LIN {X 0,Y 420.94,Z 649.275,A -85,B 0,C 180,E1 -10152.356,E2 -10152.356} C_VEL
LIN {X 0,Y 419.985,Z 659.535,A -85,B 0,C 180,E1 -10153.721,E2 -10153.721} C_VEL
LIN {X 0,Y 419.053,Z 670.297,A -85,B 0,C 180,E1 -10155.428,E2 -10155.428} C_VEL
LIN {X 0,Y 418.282,Z 678.791,A -85,B 0,C 180,E1 -10157.037,E2 -10157.037} C_VEL
LIN {X 0,Y 417.855,Z 686.7,A -85,B 0,C 180,E1 -10158.846,E2 -10158.846} C_VEL
LIN {X 0,Y 417.37,Z 693.601,A -85,B 0,C 180,E1 -10160.794,E2 -10160.794} C_VEL
LIN {X 0,Y 417.15,Z 699.002,A -85,B 0,C 180,E1 -10162.739,E2 -10162.739} C_VEL
LIN {X 0,Y 417.07,Z 702.122,A -85,B 0,C 180,E1 -10164.196,E2 -10164.196} C_VEL
LIN {X 0,Y 416.971,Z 705.164,A -85,B 0,C 180,E1 -10166.133,E2 -10166.133} C_VEL
LIN {X 0,Y 417.064,Z 706.972,A -85,B 0,C 180,E1 -10168.067,E2 -10168.067} C_VEL
LIN {X 0,Y 417.001,Z 707.573,A -85,B 0,C 180,E1 -10169.999,E2 -10169.999} C_VEL
LIN {X 0,Y 417.065,Z 706.947,A -85,B 0,C 180,E1 -10171.93,E2 -10171.93} C_VEL
LIN {X 0,Y 416.99,Z 705.073,A -85,B 0,C 180,E1 -10173.864,E2 -10173.864} C_VEL
LIN {X 0,Y 417.068,Z 701.964,A -85,B 0,C 180,E1 -10175.801,E2 -10175.801} C_VEL
LIN {X 0,Y 417.23,Z 697.54,A -85,B 0,C 180,E1 -10177.743,E2 -10177.743} C_VEL
LIN {X 0,Y 417.436,Z 691.68,A -85,B 0,C 180,E1 -10179.691,E2 -10179.691} C_VEL
LIN {X 0,Y 417.936,Z 684.237,A -85,B 0,C 180,E1 -10181.64,E2 -10181.64} C_VEL
LIN {X 0,Y 418.477,Z 676.012,A -85,B 0,C 180,E1 -10183.394,E2 -10183.394} C_VEL
LIN {X 0,Y 419.269,Z 666.599,A -85,B 0,C 180,E1 -10185.058,E2 -10185.058} C_VEL
LIN {X 0,Y 420.141,Z 656.761,A -85,B 0,C 180,E1 -10186.52,E2 -10186.52} C_VEL
LIN {X 0,Y 421.138,Z 645.151,A -85,B 0,C 180,E1 -10187.97,E2 -10187.97} C_VEL
LIN {X 0,Y 422.119,Z 633.46,A -85,B 0,C 180,E1 -10189.196,E2 -10189.196} C_VEL
LIN {X 0,Y 423.228,Z 621.023,A -85,B 0,C 180,E1 -10190.28,E2 -10190.28} C_VEL
LIN {X 0,Y 424.236,Z 607.577,A -85,B 0,C 180,E1 -10191.245,E2 -10191.245} C_VEL
LIN {X 0,Y 425.287,Z 593.073,A -85,B 0,C 180,E1 -10192.071,E2 -10192.071} C_VEL
LIN {X 0,Y 426.147,Z 577.388,A -85,B 0,C 180,E1 -10192.75,E2 -10192.75} C_VEL
LIN {X 0,Y 426.824,Z 562.272,A -85,B 0,C 180,E1 -10193.205,E2 -10193.205} C_VEL
LIN {X 0,Y 429.831,Z 427.525,A -85,B 0,C 180,E1 -10195.772,E2 -10195.772} C_VEL
LIN {X 0,Y 423.925,Z 395.924,A -85,B 0,C 180,E1 -10196.788,E2 -10196.788} C_VEL
LIN {X 0,Y 424.456,Z 389.484,A -85,B 0,C 180,E1 -10197.84,E2 -10197.84} C_VEL
LIN {X 0,Y 421.951,Z 377.843,A -85,B 0,C 180,E1 -10199.991,E2 -10199.991} C_VEL
LIN {X 0,Y 418.225,Z 363.016,A -85,B 0,C 180,E1 -10202.888,E2 -10202.888} C_VEL
LIN {X 0,Y 418.23,Z 363.015,A -85,B 0,C 180,E1 -10206.023,E2 -10206.023} C_VEL
LIN {X 0,Y 418.195,Z 363.017,A -85,B 0,C 180,E1 -10209.371,E2 -10209.371} C_VEL
LIN {X 0,Y 418.202,Z 363.019,A -85,B 0,C 180,E1 -10212.317,E2 -10212.317} C_VEL
LIN {X 0,Y 418.223,Z 363.01,A -85,B 0,C 180,E1 -10215.107,E2 -10215.107} C_VEL
LIN {X 0,Y 418.208,Z 363.015,A -85,B 0,C 180,E1 -10217.763,E2 -10217.763} C_VEL
LIN {X 0,Y 418.221,Z 363.011,A -85,B 0,C 180,E1 -10221.555,E2 -10221.555} C_VEL
LIN {X 0,Y 418.244,Z 363.007,A -85,B 0,C 180,E1 -10225.158,E2 -10225.158} C_VEL
LIN {X 0,Y 418.232,Z 363.01,A -85,B 0,C 180,E1 -10227.471,E2 -10227.471} C_VEL
LIN {X 0,Y 418.245,Z 363.008,A -85,B 0,C 180,E1 -10230.897,E2 -10230.897} C_VEL
LIN {X 0,Y 418.204,Z 363.02,A -85,B 0,C 180,E1 -10234.092,E2 -10234.092} C_VEL
LIN {X 0,Y 418.213,Z 363.011,A -85,B 0,C 180,E1 -10237.263,E2 -10237.263} C_VEL
LIN {X 0,Y 418.268,Z 363.008,A -85,B 0,C 180,E1 -10240.364,E2 -10240.364} C_VEL
LIN {X 0,Y 418.264,Z 363.006,A -85,B 0,C 180,E1 -10243.403,E2 -10243.403} C_VEL
LIN {X 0,Y 418.331,Z 362.996,A -85,B 0,C 180,E1 -10246.999,E2 -10246.999} C_VEL
LIN {X 0,Y 418.319,Z 363.002,A -85,B 0,C 180,E1 -10250.328,E2 -10250.328} C_VEL
LIN {X 0,Y 418.427,Z 362.985,A -85,B 0,C 180,E1 -10253.248,E2 -10253.248} C_VEL
LIN {X 0,Y 418.302,Z 363,A -85,B 0,C 180,E1 -10255.181,E2 -10255.181} C_VEL
LIN {X 0,Y 418.517,Z 362.98,A -85,B 0,C 180,E1 -10258.076,E2 -10258.076} C_VEL
LIN {X 0,Y 418.526,Z 362.98,A -85,B 0,C 180,E1 -10260,E2 -10260} C_VEL
LIN {X 0,Y 418.453,Z 362.981,A -85,B 0,C 180,E1 -10262.888,E2 -10262.888} C_VEL
LIN {X 0,Y 418.425,Z 362.985,A -85,B 0,C 180,E1 -10266.512,E2 -10266.512} C_VEL
LIN {X 0,Y 418.354,Z 362.994,A -85,B 0,C 180,E1 -10268.696,E2 -10268.696} C_VEL
LIN {X 0,Y 418.339,Z 362.996,A -85,B 0,C 180,E1 -10272.615,E2 -10272.615} C_VEL
LIN {X 0,Y 418.237,Z 363.011,A -85,B 0,C 180,E1 -10275.597,E2 -10275.597} C_VEL
LIN {X 0,Y 418.255,Z 363.007,A -85,B 0,C 180,E1 -10278.618,E2 -10278.618} C_VEL
LIN {X 0,Y 418.22,Z 363.015,A -85,B 0,C 180,E1 -10281.697,E2 -10281.697} C_VEL
LIN {X 0,Y 418.231,Z 363.009,A -85,B 0,C 180,E1 -10284.853,E2 -10284.853} C_VEL
LIN {X 0,Y 418.195,Z 363.019,A -85,B 0,C 180,E1 -10288.071,E2 -10288.071} C_VEL
LIN {X 0,Y 418.227,Z 363.01,A -85,B 0,C 180,E1 -10291.021,E2 -10291.021} C_VEL
LIN {X 0,Y 418.236,Z 363.013,A -85,B 0,C 180,E1 -10293.679,E2 -10293.679} C_VEL
LIN {X 0,Y 418.222,Z 363.011,A -85,B 0,C 180,E1 -10297.226,E2 -10297.226} C_VEL
LIN {X 0,Y 418.197,Z 363.013,A -85,B 0,C 180,E1 -10300.869,E2 -10300.869} C_VEL
LIN {X 0,Y 418.193,Z 363.02,A -85,B 0,C 180,E1 -10303.73,E2 -10303.73} C_VEL
LIN {X 0,Y 418.192,Z 363.015,A -85,B 0,C 180,E1 -10306.449,E2 -10306.449} C_VEL
LIN {X 0,Y 418.199,Z 363.014,A -85,B 0,C 180,E1 -10309.135,E2 -10309.135} C_VEL
LIN {X 0,Y 418.228,Z 363.009,A -85,B 0,C 180,E1 -10312.777,E2 -10312.777} C_VEL
LIN {X 0,Y 418.232,Z 363.01,A -85,B 0,C 180,E1 -10316.324,E2 -10316.324} C_VEL
LIN {X 0,Y 418.237,Z 363.015,A -85,B 0,C 180,E1 -10319.729,E2 -10319.729} C_VEL
LIN {X 0,Y 418.207,Z 363.013,A -85,B 0,C 180,E1 -10323.018,E2 -10323.018} C_VEL
LIN {X 0,Y 418.254,Z 363.008,A -85,B 0,C 180,E1 -10326.219,E2 -10326.219} C_VEL
LIN {X 0,Y 418.248,Z 363.01,A -85,B 0,C 180,E1 -10329.339,E2 -10329.339} C_VEL
LIN {X 0,Y 418.278,Z 363.004,A -85,B 0,C 180,E1 -10332.397,E2 -10332.397} C_VEL
LIN {X 0,Y 418.301,Z 363.004,A -85,B 0,C 180,E1 -10335.405,E2 -10335.405} C_VEL
LIN {X 0,Y 418.314,Z 362.999,A -85,B 0,C 180,E1 -10338.371,E2 -10338.371} C_VEL
LIN {X 0,Y 418.448,Z 362.983,A -85,B 0,C 180,E1 -10342.28,E2 -10342.28} C_VEL
LIN {X 0,Y 418.473,Z 362.98,A -85,B 0,C 180,E1 -10344.218,E2 -10344.218} C_VEL
LIN {X 0,Y 418.536,Z 362.974,A -85,B 0,C 180,E1 -10348.077,E2 -10348.077} C_VEL
LIN {X 0,Y 418.546,Z 362.973,A -85,B 0,C 180,E1 -10350.001,E2 -10350.001} C_VEL
LIN {X 0,Y 418.476,Z 362.979,A -85,B 0,C 180,E1 -10352.889,E2 -10352.889} C_VEL
LIN {X 0,Y 418.489,Z 362.983,A -85,B 0,C 180,E1 -10355.784,E2 -10355.784} C_VEL
LIN {X 0,Y 418.382,Z 362.99,A -85,B 0,C 180,E1 -10358.697,E2 -10358.697} C_VEL
LIN {X 0,Y 418.319,Z 363.006,A -85,B 0,C 180,E1 -10361.632,E2 -10361.632} C_VEL
LIN {X 0,Y 418.327,Z 363.001,A -85,B 0,C 180,E1 -10363.305,E2 -10363.305} C_VEL
LIN {X 0,Y 417.621,Z 363.094,A -85,B 0,C 180,E1 -10364.108,E2 -10364.108} C_VEL
LIN {X 0,Y 414.724,Z 363.452,A -85,B 0,C 180,E1 -10365.413,E2 -10365.413} C_VEL
LIN {X 0,Y 412.302,Z 363.748,A -85,B 0,C 180,E1 -10366.466,E2 -10366.466} C_VEL
LIN {X 0,Y 411.278,Z 363.879,A -85,B 0,C 180,E1 -10367.281,E2 -10367.281} C_VEL
LIN {X 0,Y 411.203,Z 363.885,A -85,B 0,C 180,E1 -10367.557,E2 -10367.557} C_VEL
LIN {X 0,Y 411.202,Z 363.886,A -85,B 0,C 180,E1 -10371.035,E2 -10371.035} C_VEL
LIN {X 0,Y 411.198,Z 363.886,A -85,B 0,C 180,E1 -10374.218,E2 -10374.218} C_VEL
LIN {X 0,Y 411.178,Z 363.894,A -85,B 0,C 180,E1 -10377.485,E2 -10377.485} C_VEL
LIN {X 0,Y 411.203,Z 363.89,A -85,B 0,C 180,E1 -10379.714,E2 -10379.714} C_VEL
LIN {X 0,Y 411.213,Z 363.886,A -85,B 0,C 180,E1 -10383.156,E2 -10383.156} C_VEL
LIN {X 0,Y 411.198,Z 363.891,A -85,B 0,C 180,E1 -10386.553,E2 -10386.553} C_VEL
LIN {X 0,Y 411.202,Z 363.892,A -85,B 0,C 180,E1 -10389.725,E2 -10389.725} C_VEL
LIN {X 0,Y 411.218,Z 363.936,A -85,B 0,C 180,E1 -10391.576,E2 -10391.576} C_VEL
LIN {X 0,Y 413.441,Z 373.517,A -85,B 0,C 180,E1 -10393.635,E2 -10393.635} C_VEL
LIN {X 0,Y 422.18,Z 395.363,A -85,B 0,C 180,E1 -10394.659,E2 -10394.659} C_VEL
LIN {X 0,Y 423.567,Z 402.05,A -85,B 0,C 180,E1 -10394.884,E2 -10394.884} C_VEL
LIN {X 0,Y 420.269,Z 539.555,A -85,B 0,C 180,E1 -10397.564,E2 -10397.564} C_VEL
LIN {X 0,Y 419.622,Z 555.1,A -85,B 0,C 180,E1 -10398.059,E2 -10398.059} C_VEL
LIN {X 0,Y 418.811,Z 569.926,A -85,B 0,C 180,E1 -10398.723,E2 -10398.723} C_VEL
LIN {X 0,Y 417.84,Z 584.262,A -85,B 0,C 180,E1 -10399.562,E2 -10399.562} C_VEL
LIN {X 0,Y 416.764,Z 598.407,A -85,B 0,C 180,E1 -10400.607,E2 -10400.607} C_VEL
LIN {X 0,Y 415.718,Z 611,A -85,B 0,C 180,E1 -10401.744,E2 -10401.744} C_VEL
LIN {X 0,Y 414.639,Z 623.17,A -85,B 0,C 180,E1 -10403.068,E2 -10403.068} C_VEL
LIN {X 0,Y 413.561,Z 633.744,A -85,B 0,C 180,E1 -10404.436,E2 -10404.436} C_VEL
LIN {X 0,Y 412.613,Z 644.145,A -85,B 0,C 180,E1 -10406.038,E2 -10406.038} C_VEL
LIN {X 0,Y 411.827,Z 653.503,A -85,B 0,C 180,E1 -10407.771,E2 -10407.771} C_VEL
LIN {X 0,Y 411.09,Z 662.131,A -85,B 0,C 180,E1 -10409.713,E2 -10409.713} C_VEL
LIN {X 0,Y 410.679,Z 668.101,A -85,B 0,C 180,E1 -10411.369,E2 -10411.369} C_VEL
LIN {X 0,Y 410.394,Z 672.802,A -85,B 0,C 180,E1 -10412.938,E2 -10412.938} C_VEL
LIN {X 0,Y 410.122,Z 676.864,A -85,B 0,C 180,E1 -10414.633,E2 -10414.633} C_VEL
LIN {X 0,Y 409.878,Z 680.598,A -85,B 0,C 180,E1 -10416.773,E2 -10416.773} C_VEL
LIN {X 0,Y 409.789,Z 682.843,A -85,B 0,C 180,E1 -10418.89,E2 -10418.89} C_VEL
LIN {X 0,Y 409.82,Z 683.692,A -85,B 0,C 180,E1 -10420.984,E2 -10420.984} C_VEL
LIN {X 0,Y 409.799,Z 683.207,A -85,B 0,C 180,E1 -10423.049,E2 -10423.049} C_VEL
LIN {X 0,Y 409.883,Z 681.43,A -85,B 0,C 180,E1 -10425.096,E2 -10425.096} C_VEL
LIN {X 0,Y 410.102,Z 678.363,A -85,B 0,C 180,E1 -10427.127,E2 -10427.127} C_VEL
LIN {X 0,Y 410.393,Z 673.982,A -85,B 0,C 180,E1 -10429.142,E2 -10429.142} C_VEL
LIN {X 0,Y 410.823,Z 668.208,A -85,B 0,C 180,E1 -10431.143,E2 -10431.143} C_VEL
LIN {X 0,Y 411.487,Z 660.887,A -85,B 0,C 180,E1 -10433.133,E2 -10433.133} C_VEL
LIN {X 0,Y 412.241,Z 653.05,A -85,B 0,C 180,E1 -10434.865,E2 -10434.865} C_VEL
LIN {X 0,Y 413.188,Z 643.649,A -85,B 0,C 180,E1 -10436.587,E2 -10436.587} C_VEL
LIN {X 0,Y 414.249,Z 634.122,A -85,B 0,C 180,E1 -10438.055,E2 -10438.055} C_VEL
LIN {X 0,Y 415.254,Z 623.92,A -85,B 0,C 180,E1 -10439.396,E2 -10439.396} C_VEL
LIN {X 0,Y 416.508,Z 611.806,A -85,B 0,C 180,E1 -10440.725,E2 -10440.725} C_VEL
LIN {X 0,Y 417.817,Z 598.517,A -85,B 0,C 180,E1 -10441.928,E2 -10441.928} C_VEL
LIN {X 0,Y 418.892,Z 585.618,A -85,B 0,C 180,E1 -10442.885,E2 -10442.885} C_VEL
LIN {X 0,Y 420.035,Z 570.58,A -85,B 0,C 180,E1 -10443.777,E2 -10443.777} C_VEL
LIN {X 0,Y 420.971,Z 554.73,A -85,B 0,C 180,E1 -10444.488,E2 -10444.488} C_VEL
LIN {X 0,Y 421.672,Z 539.807,A -85,B 0,C 180,E1 -10444.96,E2 -10444.96} C_VEL
LIN {X 0,Y 425.402,Z 420.585,A -85,B 0,C 180,E1 -10447.467,E2 -10447.467} C_VEL
LIN {X 0,Y 425.949,Z 402.101,A -85,B 0,C 180,E1 -10447.883,E2 -10447.883} C_VEL
LIN {X 0,Y 424.63,Z 396.844,A -85,B 0,C 180,E1 -10448.128,E2 -10448.128} C_VEL
LIN {X 0,Y 418.317,Z 383.328,A -85,B 0,C 180,E1 -10449.044,E2 -10449.044} C_VEL
LIN {X 0,Y 414.737,Z 376.273,A -85,B 0,C 180,E1 -10449.587,E2 -10449.587} C_VEL
LIN {X 0,Y 411.965,Z 366.008,A -85,B 0,C 180,E1 -10452.312,E2 -10452.312} C_VEL
LIN {X 0,Y 411.308,Z 363.875,A -85,B 0,C 180,E1 -10452.98,E2 -10452.98} C_VEL
LIN {X 0,Y 411.259,Z 363.885,A -85,B 0,C 180,E1 -10455.868,E2 -10455.868} C_VEL
LIN {X 0,Y 411.224,Z 363.887,A -85,B 0,C 180,E1 -10458.948,E2 -10458.948} C_VEL
LIN {X 0,Y 411.204,Z 363.89,A -85,B 0,C 180,E1 -10462.64,E2 -10462.64} C_VEL
LIN {X 0,Y 411.188,Z 363.889,A -85,B 0,C 180,E1 -10465.296,E2 -10465.296} C_VEL
LIN {X 0,Y 411.176,Z 363.894,A -85,B 0,C 180,E1 -10468.593,E2 -10468.593} C_VEL
LIN {X 0,Y 411.167,Z 363.895,A -85,B 0,C 180,E1 -10471.997,E2 -10471.997} C_VEL
LIN {X 0,Y 411.205,Z 363.889,A -85,B 0,C 180,E1 -10474.876,E2 -10474.876} C_VEL
LIN {X 0,Y 411.192,Z 363.893,A -85,B 0,C 180,E1 -10478.165,E2 -10478.165} C_VEL
LIN {X 0,Y 411.162,Z 363.894,A -85,B 0,C 180,E1 -10481.807,E2 -10481.807} C_VEL
LIN {X 0,Y 411.176,Z 363.891,A -85,B 0,C 180,E1 -10485.508,E2 -10485.508} C_VEL
LIN {X 0,Y 411.148,Z 363.893,A -85,B 0,C 180,E1 -10488.774,E2 -10488.774} C_VEL
LIN {X 0,Y 411.18,Z 363.895,A -85,B 0,C 180,E1 -10492.023,E2 -10492.023} C_VEL
LIN {X 0,Y 411.225,Z 363.987,A -85,B 0,C 180,E1 -10495.025,E2 -10495.025} C_VEL
LIN {X 0,Y 414.638,Z 375.681,A -85,B 0,C 180,E1 -10497.939,E2 -10497.939} C_VEL
LIN {X 0,Y 417.107,Z 385.758,A -85,B 0,C 180,E1 -10500.193,E2 -10500.193} C_VEL
LIN {X 0,Y 418.526,Z 393.484,A -85,B 0,C 180,E1 -10501.786,E2 -10501.786} C_VEL
LIN {X 0,Y 422.778,Z 413.029,A -85,B 0,C 180,E1 -10502.685,E2 -10502.685} C_VEL
LIN {X 0,Y 425.409,Z 429.771,A -85,B 0,C 180,E1 -10503.323,E2 -10503.323} C_VEL
LIN {X 0,Y 422.133,Z 535.297,A -85,B 0,C 180,E1 -10505.534,E2 -10505.534} C_VEL
LIN {X 0,Y 421.243,Z 563.028,A -85,B 0,C 180,E1 -10506.134,E2 -10506.134} C_VEL
LIN {X 0,Y 420.294,Z 578.892,A -85,B 0,C 180,E1 -10506.661,E2 -10506.661} C_VEL
LIN {X 0,Y 419.23,Z 594.331,A -85,B 0,C 180,E1 -10507.384,E2 -10507.384} C_VEL
LIN {X 0,Y 418.005,Z 609.182,A -85,B 0,C 180,E1 -10508.29,E2 -10508.29} C_VEL
LIN {X 0,Y 416.732,Z 623.432,A -85,B 0,C 180,E1 -10509.386,E2 -10509.386} C_VEL
LIN {X 0,Y 415.387,Z 636.453,A -85,B 0,C 180,E1 -10510.606,E2 -10510.606} C_VEL
LIN {X 0,Y 414.126,Z 648.749,A -85,B 0,C 180,E1 -10511.998,E2 -10511.998} C_VEL
LIN {X 0,Y 413.12,Z 659.43,A -85,B 0,C 180,E1 -10513.443,E2 -10513.443} C_VEL
LIN {X 0,Y 412.127,Z 670.174,A -85,B 0,C 180,E1 -10515.178,E2 -10515.178} C_VEL
LIN {X 0,Y 411.239,Z 679.22,A -85,B 0,C 180,E1 -10516.935,E2 -10516.935} C_VEL
LIN {X 0,Y 410.818,Z 686.549,A -85,B 0,C 180,E1 -10518.653,E2 -10518.653} C_VEL
LIN {X 0,Y 410.316,Z 693.44,A -85,B 0,C 180,E1 -10520.634,E2 -10520.634} C_VEL
LIN {X 0,Y 410.093,Z 698.83,A -85,B 0,C 180,E1 -10522.614,E2 -10522.614} C_VEL
LIN {X 0,Y 409.978,Z 701.949,A -85,B 0,C 180,E1 -10524.095,E2 -10524.095} C_VEL
LIN {X 0,Y 409.888,Z 704.98,A -85,B 0,C 180,E1 -10526.066,E2 -10526.066} C_VEL
LIN {X 0,Y 409.973,Z 706.775,A -85,B 0,C 180,E1 -10528.034,E2 -10528.034} C_VEL
LIN {X 0,Y 409.923,Z 707.359,A -85,B 0,C 180,E1 -10529.999,E2 -10529.999} C_VEL
LIN {X 0,Y 409.992,Z 706.724,A -85,B 0,C 180,E1 -10531.963,E2 -10531.963} C_VEL
LIN {X 0,Y 409.907,Z 704.826,A -85,B 0,C 180,E1 -10533.931,E2 -10533.931} C_VEL
LIN {X 0,Y 409.975,Z 701.686,A -85,B 0,C 180,E1 -10535.902,E2 -10535.902} C_VEL
LIN {X 0,Y 410.152,Z 697.225,A -85,B 0,C 180,E1 -10537.877,E2 -10537.877} C_VEL
LIN {X 0,Y 410.364,Z 691.321,A -85,B 0,C 180,E1 -10539.86,E2 -10539.86} C_VEL
LIN {X 0,Y 410.862,Z 684.865,A -85,B 0,C 180,E1 -10541.593,E2 -10541.593} C_VEL
LIN {X 0,Y 411.384,Z 676.918,A -85,B 0,C 180,E1 -10543.355,E2 -10543.355} C_VEL
LIN {X 0,Y 412.179,Z 667.579,A -85,B 0,C 180,E1 -10545.07,E2 -10545.07} C_VEL
LIN {X 0,Y 413.071,Z 657.952,A -85,B 0,C 180,E1 -10546.556,E2 -10546.556} C_VEL
LIN {X 0,Y 414.067,Z 647.023,A -85,B 0,C 180,E1 -10547.977,E2 -10547.977} C_VEL
LIN {X 0,Y 415.201,Z 633.916,A -85,B 0,C 180,E1 -10549.4,E2 -10549.4} C_VEL
LIN {X 0,Y 416.477,Z 620.032,A -85,B 0,C 180,E1 -10550.624,E2 -10550.624} C_VEL
LIN {X 0,Y 417.525,Z 606.43,A -85,B 0,C 180,E1 -10551.604,E2 -10551.604} C_VEL
LIN {X 0,Y 418.655,Z 591.799,A -85,B 0,C 180,E1 -10552.433,E2 -10552.433} C_VEL
LIN {X 0,Y 419.49,Z 576.703,A -85,B 0,C 180,E1 -10553.086,E2 -10553.086} C_VEL
LIN {X 0,Y 420.179,Z 561.93,A -85,B 0,C 180,E1 -10553.535,E2 -10553.535} C_VEL
LIN {X 0,Y 423.328,Z 428.879,A -85,B 0,C 180,E1 -10556.121,E2 -10556.121} C_VEL
LIN {X 0,Y 417.205,Z 395.591,A -85,B 0,C 180,E1 -10557.235,E2 -10557.235} C_VEL
LIN {X 0,Y 417.492,Z 390.334,A -85,B 0,C 180,E1 -10558.12,E2 -10558.12} C_VEL
LIN {X 0,Y 414.952,Z 379.016,A -85,B 0,C 180,E1 -10560.256,E2 -10560.256} C_VEL
LIN {X 0,Y 411.185,Z 363.891,A -85,B 0,C 180,E1 -10563.265,E2 -10563.265} C_VEL
LIN {X 0,Y 411.18,Z 363.891,A -85,B 0,C 180,E1 -10566.55,E2 -10566.55} C_VEL
LIN {X 0,Y 411.158,Z 363.895,A -85,B 0,C 180,E1 -10569.719,E2 -10569.719} C_VEL
LIN {X 0,Y 411.154,Z 363.891,A -85,B 0,C 180,E1 -10573.134,E2 -10573.134} C_VEL
LIN {X 0,Y 411.152,Z 363.895,A -85,B 0,C 180,E1 -10575.881,E2 -10575.881} C_VEL
LIN {X 0,Y 411.135,Z 363.894,A -85,B 0,C 180,E1 -10578.773,E2 -10578.773} C_VEL
LIN {X 0,Y 411.169,Z 363.895,A -85,B 0,C 180,E1 -10582.024,E2 -10582.024} C_VEL
LIN {X 0,Y 411.192,Z 363.888,A -85,B 0,C 180,E1 -10585.665,E2 -10585.665} C_VEL
LIN {X 0,Y 411.175,Z 363.888,A -85,B 0,C 180,E1 -10589.151,E2 -10589.151} C_VEL
LIN {X 0,Y 411.158,Z 363.891,A -85,B 0,C 180,E1 -10591.406,E2 -10591.406} C_VEL
LIN {X 0,Y 411.173,Z 363.888,A -85,B 0,C 180,E1 -10594.941,E2 -10594.941} C_VEL
LIN {X 0,Y 411.188,Z 363.891,A -85,B 0,C 180,E1 -10597.913,E2 -10597.913} C_VEL
LIN {X 0,Y 411.2,Z 363.885,A -85,B 0,C 180,E1 -10601.051,E2 -10601.051} C_VEL
LIN {X 0,Y 411.195,Z 363.892,A -85,B 0,C 180,E1 -10604.13,E2 -10604.13} C_VEL
LIN {X 0,Y 411.288,Z 363.874,A -85,B 0,C 180,E1 -10607.165,E2 -10607.165} C_VEL
LIN {X 0,Y 411.272,Z 363.882,A -85,B 0,C 180,E1 -10610.161,E2 -10610.161} C_VEL
LIN {X 0,Y 411.376,Z 363.863,A -85,B 0,C 180,E1 -10613.132,E2 -10613.132} C_VEL
LIN {X 0,Y 411.274,Z 363.876,A -85,B 0,C 180,E1 -10615.099,E2 -10615.099} C_VEL
LIN {X 0,Y 411.486,Z 363.857,A -85,B 0,C 180,E1 -10618.043,E2 -10618.043} C_VEL
LIN {X 0,Y 411.361,Z 363.865,A -85,B 0,C 180,E1 -10620.979,E2 -10620.979} C_VEL
LIN {X 0,Y 411.411,Z 363.859,A -85,B 0,C 180,E1 -10622.938,E2 -10622.938} C_VEL
LIN {X 0,Y 411.375,Z 363.864,A -85,B 0,C 180,E1 -10626.509,E2 -10626.509} C_VEL
LIN {X 0,Y 411.294,Z 363.873,A -85,B 0,C 180,E1 -10628.847,E2 -10628.847} C_VEL
LIN {X 0,Y 411.26,Z 363.883,A -85,B 0,C 180,E1 -10631.834,E2 -10631.834} C_VEL
LIN {X 0,Y 411.217,Z 363.883,A -85,B 0,C 180,E1 -10634.855,E2 -10634.855} C_VEL
LIN {X 0,Y 411.216,Z 363.89,A -85,B 0,C 180,E1 -10637.917,E2 -10637.917} C_VEL
LIN {X 0,Y 411.182,Z 363.887,A -85,B 0,C 180,E1 -10641.035,E2 -10641.035} C_VEL
LIN {X 0,Y 411.179,Z 363.891,A -85,B 0,C 180,E1 -10644.219,E2 -10644.219} C_VEL
LIN {X 0,Y 411.134,Z 363.896,A -85,B 0,C 180,E1 -10647.487,E2 -10647.487} C_VEL
LIN {X 0,Y 411.184,Z 363.892,A -85,B 0,C 180,E1 -10649.714,E2 -10649.714} C_VEL
LIN {X 0,Y 411.196,Z 363.886,A -85,B 0,C 180,E1 -10653.157,E2 -10653.157} C_VEL
LIN {X 0,Y 411.178,Z 363.888,A -85,B 0,C 180,E1 -10656.553,E2 -10656.553} C_VEL
LIN {X 0,Y 411.157,Z 363.896,A -85,B 0,C 180,E1 -10659.722,E2 -10659.722} C_VEL
LIN {X 0,Y 411.153,Z 363.891,A -85,B 0,C 180,E1 -10663.137,E2 -10663.137} C_VEL
LIN {X 0,Y 411.155,Z 363.897,A -85,B 0,C 180,E1 -10665.883,E2 -10665.883} C_VEL
LIN {X 0,Y 411.14,Z 363.892,A -85,B 0,C 180,E1 -10668.776,E2 -10668.776} C_VEL
LIN {X 0,Y 411.175,Z 363.893,A -85,B 0,C 180,E1 -10672.027,E2 -10672.027} C_VEL
LIN {X 0,Y 411.193,Z 363.892,A -85,B 0,C 180,E1 -10675.667,E2 -10675.667} C_VEL
LIN {X 0,Y 411.184,Z 363.888,A -85,B 0,C 180,E1 -10679.154,E2 -10679.154} C_VEL
LIN {X 0,Y 411.172,Z 363.892,A -85,B 0,C 180,E1 -10681.408,E2 -10681.408} C_VEL
LIN {X 0,Y 411.185,Z 363.887,A -85,B 0,C 180,E1 -10684.943,E2 -10684.943} C_VEL
LIN {X 0,Y 411.201,Z 363.89,A -85,B 0,C 180,E1 -10687.915,E2 -10687.915} C_VEL
LIN {X 0,Y 411.217,Z 363.884,A -85,B 0,C 180,E1 -10691.053,E2 -10691.053} C_VEL
LIN {X 0,Y 411.253,Z 363.881,A -85,B 0,C 180,E1 -10694.133,E2 -10694.133} C_VEL
LIN {X 0,Y 411.304,Z 363.874,A -85,B 0,C 180,E1 -10697.167,E2 -10697.167} C_VEL
LIN {X 0,Y 411.289,Z 363.876,A -85,B 0,C 180,E1 -10700.163,E2 -10700.163} C_VEL
LIN {X 0,Y 411.392,Z 363.862,A -85,B 0,C 180,E1 -10703.133,E2 -10703.133} C_VEL
LIN {X 0,Y 411.289,Z 363.875,A -85,B 0,C 180,E1 -10705.1,E2 -10705.1} C_VEL
LIN {X 0,Y 411.505,Z 363.85,A -85,B 0,C 180,E1 -10708.044,E2 -10708.044} C_VEL
LIN {X 0,Y 411.38,Z 363.863,A -85,B 0,C 180,E1 -10710.98,E2 -10710.98} C_VEL
LIN {X 0,Y 411.434,Z 363.856,A -85,B 0,C 180,E1 -10712.939,E2 -10712.939} C_VEL
LIN {X 0,Y 411.434,Z 363.86,A -85,B 0,C 180,E1 -10715.884,E2 -10715.884} C_VEL
LIN {X 0,Y 411.323,Z 363.87,A -85,B 0,C 180,E1 -10718.847,E2 -10718.847} C_VEL
LIN {X 0,Y 411.288,Z 363.879,A -85,B 0,C 180,E1 -10721.834,E2 -10721.834} C_VEL
LIN {X 0,Y 411.237,Z 363.881,A -85,B 0,C 180,E1 -10724.855,E2 -10724.855} C_VEL
LIN {X 0,Y 411.203,Z 363.885,A -85,B 0,C 180,E1 -10727.557,E2 -10727.557} C_VEL
LIN {X 0,Y 410.554,Z 363.97,A -85,B 0,C 180,E1 -10728.375,E2 -10728.375} C_VEL
LIN {X 0,Y 407.698,Z 364.329,A -85,B 0,C 180,E1 -10729.705,E2 -10729.705} C_VEL
LIN {X 0,Y 405.272,Z 364.63,A -85,B 0,C 180,E1 -10730.778,E2 -10730.778} C_VEL
LIN {X 0,Y 404.233,Z 364.76,A -85,B 0,C 180,E1 -10731.608,E2 -10731.608} C_VEL
LIN {X 0,Y 404.151,Z 364.764,A -85,B 0,C 180,E1 -10731.89,E2 -10731.89} C_VEL
LIN {X 0,Y 404.158,Z 364.766,A -85,B 0,C 180,E1 -10735.278,E2 -10735.278} C_VEL
LIN {X 0,Y 404.157,Z 364.765,A -85,B 0,C 180,E1 -10739.138,E2 -10739.138} C_VEL
LIN {X 0,Y 404.148,Z 364.763,A -85,B 0,C 180,E1 -10742.622,E2 -10742.622} C_VEL
LIN {X 0,Y 404.187,Z 364.762,A -85,B 0,C 180,E1 -10745.19,E2 -10745.19} C_VEL
LIN {X 0,Y 404.149,Z 364.768,A -85,B 0,C 180,E1 -10748.759,E2 -10748.759} C_VEL
LIN {X 0,Y 404.153,Z 364.891,A -85,B 0,C 180,E1 -10751.238,E2 -10751.238} C_VEL
LIN {X 0,Y 406.285,Z 373.81,A -85,B 0,C 180,E1 -10753.183,E2 -10753.183} C_VEL
LIN {X 0,Y 415.848,Z 397.324,A -85,B 0,C 180,E1 -10754.318,E2 -10754.318} C_VEL
LIN {X 0,Y 417.046,Z 402.798,A -85,B 0,C 180,E1 -10754.51,E2 -10754.51} C_VEL
LIN {X 0,Y 413.581,Z 539.851,A -85,B 0,C 180,E1 -10757.24,E2 -10757.24} C_VEL
LIN {X 0,Y 412.9,Z 555.592,A -85,B 0,C 180,E1 -10757.752,E2 -10757.752} C_VEL
LIN {X 0,Y 412.048,Z 570.674,A -85,B 0,C 180,E1 -10758.446,E2 -10758.446} C_VEL
LIN {X 0,Y 410.996,Z 585.358,A -85,B 0,C 180,E1 -10759.33,E2 -10759.33} C_VEL
LIN {X 0,Y 409.922,Z 599.076,A -85,B 0,C 180,E1 -10760.37,E2 -10760.37} C_VEL
LIN {X 0,Y 408.734,Z 612.327,A -85,B 0,C 180,E1 -10761.599,E2 -10761.599} C_VEL
LIN {X 0,Y 407.689,Z 623.881,A -85,B 0,C 180,E1 -10762.889,E2 -10762.889} C_VEL
LIN {X 0,Y 406.559,Z 634.828,A -85,B 0,C 180,E1 -10764.339,E2 -10764.339} C_VEL
LIN {X 0,Y 405.574,Z 645.412,A -85,B 0,C 180,E1 -10766.024,E2 -10766.024} C_VEL
LIN {X 0,Y 404.793,Z 654.199,A -85,B 0,C 180,E1 -10767.7,E2 -10767.7} C_VEL
LIN {X 0,Y 404.037,Z 662.848,A -85,B 0,C 180,E1 -10769.705,E2 -10769.705} C_VEL
LIN {X 0,Y 403.588,Z 668.748,A -85,B 0,C 180,E1 -10771.387,E2 -10771.387} C_VEL
LIN {X 0,Y 403.278,Z 673.537,A -85,B 0,C 180,E1 -10773.056,E2 -10773.056} C_VEL
LIN {X 0,Y 402.969,Z 678.068,A -85,B 0,C 180,E1 -10775.083,E2 -10775.083} C_VEL
LIN {X 0,Y 402.806,Z 680.197,A -85,B 0,C 180,E1 -10776.34,E2 -10776.34} C_VEL
LIN {X 0,Y 402.704,Z 682.717,A -85,B 0,C 180,E1 -10778.5,E2 -10778.5} C_VEL
LIN {X 0,Y 402.737,Z 683.828,A -85,B 0,C 180,E1 -10780.636,E2 -10780.636} C_VEL
LIN {X 0,Y 402.682,Z 683.599,A -85,B 0,C 180,E1 -10782.74,E2 -10782.74} C_VEL
LIN {X 0,Y 402.776,Z 682.072,A -85,B 0,C 180,E1 -10784.827,E2 -10784.827} C_VEL
LIN {X 0,Y 402.965,Z 679.256,A -85,B 0,C 180,E1 -10786.895,E2 -10786.895} C_VEL
LIN {X 0,Y 403.293,Z 675.117,A -85,B 0,C 180,E1 -10788.948,E2 -10788.948} C_VEL
LIN {X 0,Y 403.708,Z 669.602,A -85,B 0,C 180,E1 -10790.986,E2 -10790.986} C_VEL
LIN {X 0,Y 404.378,Z 662.555,A -85,B 0,C 180,E1 -10793.012,E2 -10793.012} C_VEL
LIN {X 0,Y 405.164,Z 655.04,A -85,B 0,C 180,E1 -10794.775,E2 -10794.775} C_VEL
LIN {X 0,Y 406.135,Z 646.009,A -85,B 0,C 180,E1 -10796.527,E2 -10796.527} C_VEL
LIN {X 0,Y 407.412,Z 635.125,A -85,B 0,C 180,E1 -10798.27,E2 -10798.27} C_VEL
LIN {X 0,Y 408.6,Z 623.68,A -85,B 0,C 180,E1 -10799.795,E2 -10799.795} C_VEL
LIN {X 0,Y 410.039,Z 610.579,A -85,B 0,C 180,E1 -10801.227,E2 -10801.227} C_VEL
LIN {X 0,Y 411.399,Z 597.056,A -85,B 0,C 180,E1 -10802.447,E2 -10802.447} C_VEL
LIN {X 0,Y 412.598,Z 583.867,A -85,B 0,C 180,E1 -10803.418,E2 -10803.418} C_VEL
LIN {X 0,Y 413.71,Z 569.46,A -85,B 0,C 180,E1 -10804.262,E2 -10804.262} C_VEL
LIN {X 0,Y 414.635,Z 553.944,A -85,B 0,C 180,E1 -10804.953,E2 -10804.953} C_VEL
LIN {X 0,Y 415.376,Z 538.501,A -85,B 0,C 180,E1 -10805.431,E2 -10805.431} C_VEL
LIN {X 0,Y 419.277,Z 423.67,A -85,B 0,C 180,E1 -10807.906,E2 -10807.906} C_VEL
LIN {X 0,Y 419.998,Z 403.904,A -85,B 0,C 180,E1 -10808.35,E2 -10808.35} C_VEL
LIN {X 0,Y 418.921,Z 399.845,A -85,B 0,C 180,E1 -10808.549,E2 -10808.549} C_VEL
LIN {X 0,Y 413.107,Z 387.213,A -85,B 0,C 180,E1 -10809.437,E2 -10809.437} C_VEL
LIN {X 0,Y 407.601,Z 376.64,A -85,B 0,C 180,E1 -10810.314,E2 -10810.314} C_VEL
LIN {X 0,Y 404.865,Z 366.854,A -85,B 0,C 180,E1 -10813.042,E2 -10813.042} C_VEL
LIN {X 0,Y 404.229,Z 364.761,A -85,B 0,C 180,E1 -10813.735,E2 -10813.735} C_VEL
LIN {X 0,Y 404.208,Z 364.763,A -85,B 0,C 180,E1 -10817.192,E2 -10817.192} C_VEL
LIN {X 0,Y 404.169,Z 364.767,A -85,B 0,C 180,E1 -10820.351,E2 -10820.351} C_VEL
LIN {X 0,Y 404.154,Z 364.768,A -85,B 0,C 180,E1 -10823.575,E2 -10823.575} C_VEL
LIN {X 0,Y 404.109,Z 364.773,A -85,B 0,C 180,E1 -10826.883,E2 -10826.883} C_VEL
LIN {X 0,Y 404.146,Z 364.77,A -85,B 0,C 180,E1 -10830.285,E2 -10830.285} C_VEL
LIN {X 0,Y 404.141,Z 364.77,A -85,B 0,C 180,E1 -10833.812,E2 -10833.812} C_VEL
LIN {X 0,Y 404.134,Z 364.769,A -85,B 0,C 180,E1 -10836.873,E2 -10836.873} C_VEL
LIN {X 0,Y 404.121,Z 364.772,A -85,B 0,C 180,E1 -10840.074,E2 -10840.074} C_VEL
LIN {X 0,Y 404.143,Z 364.766,A -85,B 0,C 180,E1 -10843.081,E2 -10843.081} C_VEL
LIN {X 0,Y 404.123,Z 364.77,A -85,B 0,C 180,E1 -10845.921,E2 -10845.921} C_VEL
LIN {X 0,Y 404.103,Z 364.771,A -85,B 0,C 180,E1 -10848.632,E2 -10848.632} C_VEL
LIN {X 0,Y 404.136,Z 364.77,A -85,B 0,C 180,E1 -10851.495,E2 -10851.495} C_VEL
LIN {X 0,Y 404.156,Z 364.913,A -85,B 0,C 180,E1 -10854.294,E2 -10854.294} C_VEL
LIN {X 0,Y 407.365,Z 375.495,A -85,B 0,C 180,E1 -10857.081,E2 -10857.081} C_VEL
LIN {X 0,Y 409.882,Z 385.204,A -85,B 0,C 180,E1 -10859.376,E2 -10859.376} C_VEL
LIN {X 0,Y 411.663,Z 393.587,A -85,B 0,C 180,E1 -10861.154,E2 -10861.154} C_VEL
LIN {X 0,Y 413.251,Z 398.07,A -85,B 0,C 180,E1 -10861.431,E2 -10861.431} C_VEL
LIN {X 0,Y 417.178,Z 416.841,A -85,B 0,C 180,E1 -10862.298,E2 -10862.298} C_VEL
LIN {X 0,Y 419.34,Z 430.765,A -85,B 0,C 180,E1 -10862.838,E2 -10862.838} C_VEL
LIN {X 0,Y 415.755,Z 537.237,A -85,B 0,C 180,E1 -10865.133,E2 -10865.133} C_VEL
LIN {X 0,Y 414.859,Z 563.224,A -85,B 0,C 180,E1 -10865.71,E2 -10865.71} C_VEL
LIN {X 0,Y 413.787,Z 579.723,A -85,B 0,C 180,E1 -10866.276,E2 -10866.276} C_VEL
LIN {X 0,Y 412.71,Z 594.645,A -85,B 0,C 180,E1 -10866.999,E2 -10866.999} C_VEL
LIN {X 0,Y 411.415,Z 609.421,A -85,B 0,C 180,E1 -10867.924,E2 -10867.924} C_VEL
LIN {X 0,Y 410.083,Z 623.532,A -85,B 0,C 180,E1 -10869.036,E2 -10869.036} C_VEL
LIN {X 0,Y 408.676,Z 636.486,A -85,B 0,C 180,E1 -10870.275,E2 -10870.275} C_VEL
LIN {X 0,Y 407.397,Z 648.422,A -85,B 0,C 180,E1 -10871.65,E2 -10871.65} C_VEL
LIN {X 0,Y 406.277,Z 659.372,A -85,B 0,C 180,E1 -10873.156,E2 -10873.156} C_VEL
LIN {X 0,Y 405.202,Z 670.083,A -85,B 0,C 180,E1 -10874.919,E2 -10874.919} C_VEL
LIN {X 0,Y 404.383,Z 678.068,A -85,B 0,C 180,E1 -10876.48,E2 -10876.48} C_VEL
LIN {X 0,Y 403.897,Z 684.451,A -85,B 0,C 180,E1 -10877.946,E2 -10877.946} C_VEL
LIN {X 0,Y 403.479,Z 690.054,A -85,B 0,C 180,E1 -10879.46,E2 -10879.46} C_VEL
LIN {X 0,Y 403.119,Z 696.159,A -85,B 0,C 180,E1 -10881.477,E2 -10881.477} C_VEL
LIN {X 0,Y 402.976,Z 699.793,A -85,B 0,C 180,E1 -10882.986,E2 -10882.986} C_VEL
LIN {X 0,Y 402.857,Z 703.453,A -85,B 0,C 180,E1 -10884.994,E2 -10884.994} C_VEL
LIN {X 0,Y 402.803,Z 705.843,A -85,B 0,C 180,E1 -10886.998,E2 -10886.998} C_VEL
LIN {X 0,Y 402.862,Z 707.013,A -85,B 0,C 180,E1 -10888.999,E2 -10888.999} C_VEL
LIN {X 0,Y 402.862,Z 706.974,A -85,B 0,C 180,E1 -10890.998,E2 -10890.998} C_VEL
LIN {X 0,Y 402.902,Z 706.493,A -85,B 0,C 180,E1 -10891.998,E2 -10891.998} C_VEL
LIN {X 0,Y 402.826,Z 704.571,A -85,B 0,C 180,E1 -10894,E2 -10894} C_VEL
LIN {X 0,Y 402.897,Z 701.173,A -85,B 0,C 180,E1 -10896.128,E2 -10896.128} C_VEL
LIN {X 0,Y 403.069,Z 696.894,A -85,B 0,C 180,E1 -10898.017,E2 -10898.017} C_VEL
LIN {X 0,Y 403.303,Z 690.942,A -85,B 0,C 180,E1 -10900.034,E2 -10900.034} C_VEL
LIN {X 0,Y 403.795,Z 684.432,A -85,B 0,C 180,E1 -10901.799,E2 -10901.799} C_VEL
LIN {X 0,Y 404.354,Z 676.792,A -85,B 0,C 180,E1 -10903.518,E2 -10903.518} C_VEL
LIN {X 0,Y 405.242,Z 667.018,A -85,B 0,C 180,E1 -10905.334,E2 -10905.334} C_VEL
LIN {X 0,Y 406.178,Z 657.313,A -85,B 0,C 180,E1 -10906.846,E2 -10906.846} C_VEL
LIN {X 0,Y 407.256,Z 645.769,A -85,B 0,C 180,E1 -10908.354,E2 -10908.354} C_VEL
LIN {X 0,Y 408.422,Z 633.041,A -85,B 0,C 180,E1 -10909.735,E2 -10909.735} C_VEL
LIN {X 0,Y 409.602,Z 620.584,A -85,B 0,C 180,E1 -10910.855,E2 -10910.855} C_VEL
LIN {X 0,Y 410.686,Z 607.125,A -85,B 0,C 180,E1 -10911.85,E2 -10911.85} C_VEL
LIN {X 0,Y 411.802,Z 592.956,A -85,B 0,C 180,E1 -10912.682,E2 -10912.682} C_VEL
LIN {X 0,Y 412.761,Z 577.279,A -85,B 0,C 180,E1 -10913.385,E2 -10913.385} C_VEL
LIN {X 0,Y 413.527,Z 561.656,A -85,B 0,C 180,E1 -10913.87,E2 -10913.87} C_VEL
LIN {X 0,Y 416.734,Z 429.364,A -85,B 0,C 180,E1 -10916.502,E2 -10916.502} C_VEL
LIN {X 0,Y 410.498,Z 395.619,A -85,B 0,C 180,E1 -10917.635,E2 -10917.635} C_VEL
LIN {X 0,Y 410.561,Z 391.442,A -85,B 0,C 180,E1 -10918.359,E2 -10918.359} C_VEL
LIN {X 0,Y 407.434,Z 377.954,A -85,B 0,C 180,E1 -10920.964,E2 -10920.964} C_VEL
LIN {X 0,Y 404.16,Z 364.766,A -85,B 0,C 180,E1 -10923.628,E2 -10923.628} C_VEL
LIN {X 0,Y 404.123,Z 364.771,A -85,B 0,C 180,E1 -10926.873,E2 -10926.873} C_VEL
LIN {X 0,Y 404.107,Z 364.775,A -85,B 0,C 180,E1 -10930.073,E2 -10930.073} C_VEL
LIN {X 0,Y 404.133,Z 364.765,A -85,B 0,C 180,E1 -10933.081,E2 -10933.081} C_VEL
LIN {X 0,Y 404.133,Z 364.769,A -85,B 0,C 180,E1 -10935.924,E2 -10935.924} C_VEL
LIN {X 0,Y 404.09,Z 364.773,A -85,B 0,C 180,E1 -10938.632,E2 -10938.632} C_VEL
LIN {X 0,Y 404.125,Z 364.767,A -85,B 0,C 180,E1 -10941.494,E2 -10941.494} C_VEL
LIN {X 0,Y 404.17,Z 364.761,A -85,B 0,C 180,E1 -10944.983,E2 -10944.983} C_VEL
LIN {X 0,Y 404.126,Z 364.77,A -85,B 0,C 180,E1 -10948.441,E2 -10948.441} C_VEL
LIN {X 0,Y 404.135,Z 364.765,A -85,B 0,C 180,E1 -10950.862,E2 -10950.862} C_VEL
LIN {X 0,Y 404.138,Z 364.766,A -85,B 0,C 180,E1 -10954.722,E2 -10954.722} C_VEL
LIN {X 0,Y 404.152,Z 364.764,A -85,B 0,C 180,E1 -10957.507,E2 -10957.507} C_VEL
LIN {X 0,Y 404.145,Z 364.765,A -85,B 0,C 180,E1 -10960.707,E2 -10960.707} C_VEL
LIN {X 0,Y 404.166,Z 364.766,A -85,B 0,C 180,E1 -10963.846,E2 -10963.846} C_VEL
LIN {X 0,Y 404.268,Z 364.748,A -85,B 0,C 180,E1 -10966.939,E2 -10966.939} C_VEL
LIN {X 0,Y 404.238,Z 364.759,A -85,B 0,C 180,E1 -10969.988,E2 -10969.988} C_VEL
LIN {X 0,Y 404.326,Z 364.741,A -85,B 0,C 180,E1 -10973.012,E2 -10973.012} C_VEL
LIN {X 0,Y 404.246,Z 364.751,A -85,B 0,C 180,E1 -10975.013,E2 -10975.013} C_VEL
LIN {X 0,Y 404.455,Z 364.733,A -85,B 0,C 180,E1 -10978.009,E2 -10978.009} C_VEL
LIN {X 0,Y 404.331,Z 364.741,A -85,B 0,C 180,E1 -10980.996,E2 -10980.996} C_VEL
LIN {X 0,Y 404.371,Z 364.736,A -85,B 0,C 180,E1 -10982.989,E2 -10982.989} C_VEL
LIN {X 0,Y 404.327,Z 364.743,A -85,B 0,C 180,E1 -10986.505,E2 -10986.505} C_VEL
LIN {X 0,Y 404.243,Z 364.752,A -85,B 0,C 180,E1 -10989.002,E2 -10989.002} C_VEL
LIN {X 0,Y 404.234,Z 364.759,A -85,B 0,C 180,E1 -10992.042,E2 -10992.042} C_VEL
LIN {X 0,Y 404.161,Z 364.762,A -85,B 0,C 180,E1 -10995.12,E2 -10995.12} C_VEL
LIN {X 0,Y 404.18,Z 364.763,A -85,B 0,C 180,E1 -10998.24,E2 -10998.24} C_VEL
LIN {X 0,Y 404.124,Z 364.768,A -85,B 0,C 180,E1 -11001.421,E2 -11001.421} C_VEL
LIN {X 0,Y 404.123,Z 364.767,A -85,B 0,C 180,E1 -11004.67,E2 -11004.67} C_VEL
LIN {X 0,Y 404.091,Z 364.776,A -85,B 0,C 180,E1 -11008.008,E2 -11008.008} C_VEL
LIN {X 0,Y 404.132,Z 364.768,A -85,B 0,C 180,E1 -11010.287,E2 -11010.287} C_VEL
LIN {X 0,Y 404.133,Z 364.772,A -85,B 0,C 180,E1 -11013.814,E2 -11013.814} C_VEL
LIN {X 0,Y 404.12,Z 364.767,A -85,B 0,C 180,E1 -11016.875,E2 -11016.875} C_VEL
LIN {X 0,Y 404.107,Z 364.773,A -85,B 0,C 180,E1 -11020.076,E2 -11020.076} C_VEL
LIN {X 0,Y 404.133,Z 364.766,A -85,B 0,C 180,E1 -11023.083,E2 -11023.083} C_VEL
LIN {X 0,Y 404.112,Z 364.774,A -85,B 0,C 180,E1 -11025.924,E2 -11025.924} C_VEL
LIN {X 0,Y 404.094,Z 364.77,A -85,B 0,C 180,E1 -11028.634,E2 -11028.634} C_VEL
LIN {X 0,Y 404.131,Z 364.769,A -85,B 0,C 180,E1 -11031.497,E2 -11031.497} C_VEL
LIN {X 0,Y 404.17,Z 364.761,A -85,B 0,C 180,E1 -11034.985,E2 -11034.985} C_VEL
LIN {X 0,Y 404.134,Z 364.766,A -85,B 0,C 180,E1 -11038.444,E2 -11038.444} C_VEL
LIN {X 0,Y 404.147,Z 364.764,A -85,B 0,C 180,E1 -11040.864,E2 -11040.864} C_VEL
LIN {X 0,Y 404.15,Z 364.763,A -85,B 0,C 180,E1 -11044.724,E2 -11044.724} C_VEL
LIN {X 0,Y 404.164,Z 364.766,A -85,B 0,C 180,E1 -11047.51,E2 -11047.51} C_VEL
LIN {X 0,Y 404.161,Z 364.762,A -85,B 0,C 180,E1 -11050.709,E2 -11050.709} C_VEL
LIN {X 0,Y 404.22,Z 364.76,A -85,B 0,C 180,E1 -11053.85,E2 -11053.85} C_VEL
LIN {X 0,Y 404.284,Z 364.747,A -85,B 0,C 180,E1 -11056.941,E2 -11056.941} C_VEL
LIN {X 0,Y 404.255,Z 364.754,A -85,B 0,C 180,E1 -11059.99,E2 -11059.99} C_VEL
LIN {X 0,Y 404.342,Z 364.74,A -85,B 0,C 180,E1 -11063.013,E2 -11063.013} C_VEL
LIN {X 0,Y 404.26,Z 364.75,A -85,B 0,C 180,E1 -11065.015,E2 -11065.015} C_VEL
LIN {X 0,Y 404.474,Z 364.726,A -85,B 0,C 180,E1 -11068.01,E2 -11068.01} C_VEL
LIN {X 0,Y 404.351,Z 364.739,A -85,B 0,C 180,E1 -11070.997,E2 -11070.997} C_VEL
LIN {X 0,Y 404.394,Z 364.734,A -85,B 0,C 180,E1 -11072.99,E2 -11072.99} C_VEL
LIN {X 0,Y 404.382,Z 364.737,A -85,B 0,C 180,E1 -11075.987,E2 -11075.987} C_VEL
LIN {X 0,Y 404.27,Z 364.749,A -85,B 0,C 180,E1 -11079.003,E2 -11079.003} C_VEL
LIN {X 0,Y 404.261,Z 364.752,A -85,B 0,C 180,E1 -11082.043,E2 -11082.043} C_VEL
LIN {X 0,Y 404.182,Z 364.761,A -85,B 0,C 180,E1 -11085.12,E2 -11085.12} C_VEL
LIN {X 0,Y 404.172,Z 364.761,A -85,B 0,C 180,E1 -11088.241,E2 -11088.241} C_VEL
LIN {X 0,Y 404.165,Z 364.767,A -85,B 0,C 180,E1 -11091.419,E2 -11091.419} C_VEL
LIN {X 0,Y 404.151,Z 364.764,A -85,B 0,C 180,E1 -11091.89,E2 -11091.89} C_VEL
LIN {X 0,Y 403.495,Z 364.845,A -85,B 0,C 180,E1 -11092.721,E2 -11092.721} C_VEL
LIN {X 0,Y 400.659,Z 365.2,A -85,B 0,C 180,E1 -11094.072,E2 -11094.072} C_VEL
LIN {X 0,Y 398.24,Z 365.502,A -85,B 0,C 180,E1 -11095.163,E2 -11095.163} C_VEL
LIN {X 0,Y 397.181,Z 365.634,A -85,B 0,C 180,E1 -11096.007,E2 -11096.007} C_VEL
LIN {X 0,Y 397.085,Z 365.644,A -85,B 0,C 180,E1 -11096.293,E2 -11096.293} C_VEL
LIN {X 0,Y 397.105,Z 365.644,A -85,B 0,C 180,E1 -11099.864,E2 -11099.864} C_VEL
LIN {X 0,Y 397.125,Z 365.643,A -85,B 0,C 180,E1 -11103.719,E2 -11103.719} C_VEL
LIN {X 0,Y 397.097,Z 365.649,A -85,B 0,C 180,E1 -11107.209,E2 -11107.209} C_VEL
LIN {X 0,Y 397.127,Z 365.651,A -85,B 0,C 180,E1 -11110.849,E2 -11110.849} C_VEL
LIN {X 0,Y 399.043,Z 373.892,A -85,B 0,C 180,E1 -11112.694,E2 -11112.694} C_VEL
LIN {X 0,Y 409.645,Z 399.923,A -85,B 0,C 180,E1 -11113.988,E2 -11113.988} C_VEL
LIN {X 0,Y 410.505,Z 404.331,A -85,B 0,C 180,E1 -11114.139,E2 -11114.139} C_VEL
LIN {X 0,Y 406.927,Z 539.887,A -85,B 0,C 180,E1 -11116.899,E2 -11116.899} C_VEL
LIN {X 0,Y 406.263,Z 555.239,A -85,B 0,C 180,E1 -11117.403,E2 -11117.403} C_VEL
LIN {X 0,Y 405.352,Z 570.389,A -85,B 0,C 180,E1 -11118.103,E2 -11118.103} C_VEL
LIN {X 0,Y 404.305,Z 584.965,A -85,B 0,C 180,E1 -11118.988,E2 -11118.988} C_VEL
LIN {X 0,Y 403.194,Z 598.582,A -85,B 0,C 180,E1 -11120.025,E2 -11120.025} C_VEL
LIN {X 0,Y 402.055,Z 610.944,A -85,B 0,C 180,E1 -11121.168,E2 -11121.168} C_VEL
LIN {X 0,Y 400.833,Z 623.875,A -85,B 0,C 180,E1 -11122.62,E2 -11122.62} C_VEL
LIN {X 0,Y 399.717,Z 634.059,A -85,B 0,C 180,E1 -11123.98,E2 -11123.98} C_VEL
LIN {X 0,Y 398.68,Z 644.634,A -85,B 0,C 180,E1 -11125.66,E2 -11125.66} C_VEL
LIN {X 0,Y 397.828,Z 653.729,A -85,B 0,C 180,E1 -11127.397,E2 -11127.397} C_VEL
LIN {X 0,Y 397.034,Z 662.424,A -85,B 0,C 180,E1 -11129.409,E2 -11129.409} C_VEL
LIN {X 0,Y 396.51,Z 669.36,A -85,B 0,C 180,E1 -11131.408,E2 -11131.408} C_VEL
LIN {X 0,Y 396.177,Z 674.057,A -85,B 0,C 180,E1 -11133.105,E2 -11133.105} C_VEL
LIN {X 0,Y 395.897,Z 677.975,A -85,B 0,C 180,E1 -11134.873,E2 -11134.873} C_VEL
LIN {X 0,Y 395.686,Z 681.364,A -85,B 0,C 180,E1 -11136.998,E2 -11136.998} C_VEL
LIN {X 0,Y 395.582,Z 683.446,A -85,B 0,C 180,E1 -11139.186,E2 -11139.186} C_VEL
LIN {X 0,Y 395.593,Z 684.144,A -85,B 0,C 180,E1 -11141.35,E2 -11141.35} C_VEL
LIN {X 0,Y 395.617,Z 683.429,A -85,B 0,C 180,E1 -11143.598,E2 -11143.598} C_VEL
LIN {X 0,Y 395.736,Z 681.556,A -85,B 0,C 180,E1 -11145.603,E2 -11145.603} C_VEL
LIN {X 0,Y 396.036,Z 678.297,A -85,B 0,C 180,E1 -11147.704,E2 -11147.704} C_VEL
LIN {X 0,Y 396.357,Z 673.723,A -85,B 0,C 180,E1 -11149.786,E2 -11149.786} C_VEL
LIN {X 0,Y 396.937,Z 667.745,A -85,B 0,C 180,E1 -11151.857,E2 -11151.857} C_VEL
LIN {X 0,Y 397.726,Z 660.214,A -85,B 0,C 180,E1 -11153.914,E2 -11153.914} C_VEL
LIN {X 0,Y 398.619,Z 652.147,A -85,B 0,C 180,E1 -11155.702,E2 -11155.702} C_VEL
LIN {X 0,Y 399.734,Z 642.484,A -85,B 0,C 180,E1 -11157.481,E2 -11157.481} C_VEL
LIN {X 0,Y 400.868,Z 632.652,A -85,B 0,C 180,E1 -11158.995,E2 -11158.995} C_VEL
LIN {X 0,Y 402.305,Z 621.008,A -85,B 0,C 180,E1 -11160.5,E2 -11160.5} C_VEL
LIN {X 0,Y 403.762,Z 608.236,A -85,B 0,C 180,E1 -11161.87,E2 -11161.87} C_VEL
LIN {X 0,Y 405.042,Z 595.687,A -85,B 0,C 180,E1 -11162.984,E2 -11162.984} C_VEL
LIN {X 0,Y 406.336,Z 582.073,A -85,B 0,C 180,E1 -11163.967,E2 -11163.967} C_VEL
LIN {X 0,Y 407.395,Z 568.339,A -85,B 0,C 180,E1 -11164.762,E2 -11164.762} C_VEL
LIN {X 0,Y 408.426,Z 552.425,A -85,B 0,C 180,E1 -11165.461,E2 -11165.461} C_VEL
LIN {X 0,Y 409.169,Z 536.381,A -85,B 0,C 180,E1 -11165.946,E2 -11165.946} C_VEL
LIN {X 0,Y 412.739,Z 436.595,A -85,B 0,C 180,E1 -11168.144,E2 -11168.144} C_VEL
LIN {X 0,Y 414.011,Z 405.067,A -85,B 0,C 180,E1 -11168.868,E2 -11168.868} C_VEL
LIN {X 0,Y 412.537,Z 401.035,A -85,B 0,C 180,E1 -11169.117,E2 -11169.117} C_VEL
LIN {X 0,Y 406.647,Z 388.501,A -85,B 0,C 180,E1 -11170.054,E2 -11170.054} C_VEL
LIN {X 0,Y 400.5,Z 377.045,A -85,B 0,C 180,E1 -11171.083,E2 -11171.083} C_VEL
LIN {X 0,Y 397.925,Z 367.997,A -85,B 0,C 180,E1 -11173.735,E2 -11173.735} C_VEL
LIN {X 0,Y 397.162,Z 365.642,A -85,B 0,C 180,E1 -11174.54,E2 -11174.54} C_VEL
LIN {X 0,Y 397.149,Z 365.643,A -85,B 0,C 180,E1 -11177.507,E2 -11177.507} C_VEL
LIN {X 0,Y 397.108,Z 365.647,A -85,B 0,C 180,E1 -11180.729,E2 -11180.729} C_VEL
LIN {X 0,Y 397.112,Z 365.645,A -85,B 0,C 180,E1 -11184.019,E2 -11184.019} C_VEL
LIN {X 0,Y 397.07,Z 365.65,A -85,B 0,C 180,E1 -11187.399,E2 -11187.399} C_VEL
LIN {X 0,Y 397.101,Z 365.645,A -85,B 0,C 180,E1 -11189.862,E2 -11189.862} C_VEL
LIN {X 0,Y 397.116,Z 365.643,A -85,B 0,C 180,E1 -11193.273,E2 -11193.273} C_VEL
LIN {X 0,Y 397.096,Z 365.646,A -85,B 0,C 180,E1 -11196.995,E2 -11196.995} C_VEL
LIN {X 0,Y 397.058,Z 365.65,A -85,B 0,C 180,E1 -11200.437,E2 -11200.437} C_VEL
LIN {X 0,Y 397.089,Z 365.645,A -85,B 0,C 180,E1 -11203.65,E2 -11203.65} C_VEL
LIN {X 0,Y 397.093,Z 365.645,A -85,B 0,C 180,E1 -11206.522,E2 -11206.522} C_VEL
LIN {X 0,Y 397.087,Z 365.648,A -85,B 0,C 180,E1 -11210.418,E2 -11210.418} C_VEL
LIN {X 0,Y 397.132,Z 365.8,A -85,B 0,C 180,E1 -11213.482,E2 -11213.482} C_VEL
LIN {X 0,Y 400.418,Z 376.464,A -85,B 0,C 180,E1 -11216.456,E2 -11216.456} C_VEL
LIN {X 0,Y 403.148,Z 386.936,A -85,B 0,C 180,E1 -11219.033,E2 -11219.033} C_VEL
LIN {X 0,Y 404.494,Z 393.161,A -85,B 0,C 180,E1 -11220.407,E2 -11220.407} C_VEL
LIN {X 0,Y 407.562,Z 400.303,A -85,B 0,C 180,E1 -11220.93,E2 -11220.93} C_VEL
LIN {X 0,Y 411.326,Z 418.657,A -85,B 0,C 180,E1 -11221.803,E2 -11221.803} C_VEL
LIN {X 0,Y 413.297,Z 431.553,A -85,B 0,C 180,E1 -11222.331,E2 -11222.331} C_VEL
LIN {X 0,Y 409.528,Z 536.954,A -85,B 0,C 180,E1 -11224.661,E2 -11224.661} C_VEL
LIN {X 0,Y 408.51,Z 563.494,A -85,B 0,C 180,E1 -11225.273,E2 -11225.273} C_VEL
LIN {X 0,Y 407.336,Z 580.375,A -85,B 0,C 180,E1 -11225.873,E2 -11225.873} C_VEL
LIN {X 0,Y 406.154,Z 595.719,A -85,B 0,C 180,E1 -11226.641,E2 -11226.641} C_VEL
LIN {X 0,Y 404.849,Z 609.758,A -85,B 0,C 180,E1 -11227.547,E2 -11227.547} C_VEL
LIN {X 0,Y 403.443,Z 623.765,A -85,B 0,C 180,E1 -11228.675,E2 -11228.675} C_VEL
LIN {X 0,Y 401.97,Z 636.599,A -85,B 0,C 180,E1 -11229.931,E2 -11229.931} C_VEL
LIN {X 0,Y 400.688,Z 648.125,A -85,B 0,C 180,E1 -11231.289,E2 -11231.289} C_VEL
LIN {X 0,Y 399.435,Z 659.353,A -85,B 0,C 180,E1 -11232.858,E2 -11232.858} C_VEL
LIN {X 0,Y 398.289,Z 670.024,A -85,B 0,C 180,E1 -11234.651,E2 -11234.651} C_VEL
LIN {X 0,Y 397.33,Z 678.911,A -85,B 0,C 180,E1 -11236.444,E2 -11236.444} C_VEL
LIN {X 0,Y 396.755,Z 686.308,A -85,B 0,C 180,E1 -11238.245,E2 -11238.245} C_VEL
LIN {X 0,Y 396.193,Z 693.163,A -85,B 0,C 180,E1 -11240.297,E2 -11240.297} C_VEL
LIN {X 0,Y 395.939,Z 698.524,A -85,B 0,C 180,E1 -11242.348,E2 -11242.348} C_VEL
LIN {X 0,Y 395.82,Z 701.631,A -85,B 0,C 180,E1 -11243.883,E2 -11243.883} C_VEL
LIN {X 0,Y 395.731,Z 704.63,A -85,B 0,C 180,E1 -11245.925,E2 -11245.925} C_VEL
LIN {X 0,Y 395.766,Z 706.386,A -85,B 0,C 180,E1 -11247.963,E2 -11247.963} C_VEL
LIN {X 0,Y 395.775,Z 706.928,A -85,B 0,C 180,E1 -11249.998,E2 -11249.998} C_VEL
LIN {X 0,Y 395.799,Z 706.254,A -85,B 0,C 180,E1 -11252.034,E2 -11252.034} C_VEL
LIN {X 0,Y 395.747,Z 704.31,A -85,B 0,C 180,E1 -11254.072,E2 -11254.072} C_VEL
LIN {X 0,Y 395.818,Z 701.098,A -85,B 0,C 180,E1 -11256.114,E2 -11256.114} C_VEL
LIN {X 0,Y 395.982,Z 696.551,A -85,B 0,C 180,E1 -11258.161,E2 -11258.161} C_VEL
LIN {X 0,Y 396.245,Z 690.548,A -85,B 0,C 180,E1 -11260.215,E2 -11260.215} C_VEL
LIN {X 0,Y 396.746,Z 683.978,A -85,B 0,C 180,E1 -11262.012,E2 -11262.012} C_VEL
LIN {X 0,Y 397.388,Z 676.016,A -85,B 0,C 180,E1 -11263.811,E2 -11263.811} C_VEL
LIN {X 0,Y 398.287,Z 666.412,A -85,B 0,C 180,E1 -11265.609,E2 -11265.609} C_VEL
LIN {X 0,Y 399.28,Z 656.613,A -85,B 0,C 180,E1 -11267.145,E2 -11267.145} C_VEL
LIN {X 0,Y 400.412,Z 645.171,A -85,B 0,C 180,E1 -11268.654,E2 -11268.654} C_VEL
LIN {X 0,Y 401.522,Z 633.417,A -85,B 0,C 180,E1 -11269.955,E2 -11269.955} C_VEL
LIN {X 0,Y 402.878,Z 619.489,A -85,B 0,C 180,E1 -11271.22,E2 -11271.22} C_VEL
LIN {X 0,Y 404.04,Z 605.849,A -85,B 0,C 180,E1 -11272.228,E2 -11272.228} C_VEL
LIN {X 0,Y 405.193,Z 591.708,A -85,B 0,C 180,E1 -11273.058,E2 -11273.058} C_VEL
LIN {X 0,Y 406.082,Z 576.906,A -85,B 0,C 180,E1 -11273.725,E2 -11273.725} C_VEL
LIN {X 0,Y 406.888,Z 561.23,A -85,B 0,C 180,E1 -11274.217,E2 -11274.217} C_VEL
LIN {X 0,Y 410.206,Z 430.31,A -85,B 0,C 180,E1 -11276.878,E2 -11276.878} C_VEL
LIN {X 0,Y 403.777,Z 395.306,A -85,B 0,C 180,E1 -11278.1,E2 -11278.1} C_VEL
LIN {X 0,Y 403.327,Z 391.337,A -85,B 0,C 180,E1 -11278.836,E2 -11278.836} C_VEL
LIN {X 0,Y 399.741,Z 376.231,A -85,B 0,C 180,E1 -11281.831,E2 -11281.831} C_VEL
LIN {X 0,Y 397.116,Z 365.646,A -85,B 0,C 180,E1 -11284.059,E2 -11284.059} C_VEL
LIN {X 0,Y 397.079,Z 365.648,A -85,B 0,C 180,E1 -11287.206,E2 -11287.206} C_VEL
LIN {X 0,Y 397.045,Z 365.653,A -85,B 0,C 180,E1 -11290.436,E2 -11290.436} C_VEL
LIN {X 0,Y 397.087,Z 365.645,A -85,B 0,C 180,E1 -11293.648,E2 -11293.648} C_VEL
LIN {X 0,Y 397.085,Z 365.646,A -85,B 0,C 180,E1 -11296.521,E2 -11296.521} C_VEL
LIN {X 0,Y 397.073,Z 365.649,A -85,B 0,C 180,E1 -11300.418,E2 -11300.418} C_VEL
LIN {X 0,Y 397.081,Z 365.644,A -85,B 0,C 180,E1 -11303.003,E2 -11303.003} C_VEL
LIN {X 0,Y 397.105,Z 365.646,A -85,B 0,C 180,E1 -11306.281,E2 -11306.281} C_VEL
LIN {X 0,Y 397.085,Z 365.651,A -85,B 0,C 180,E1 -11310.136,E2 -11310.136} C_VEL
LIN {X 0,Y 397.06,Z 365.649,A -85,B 0,C 180,E1 -11313.737,E2 -11313.737} C_VEL
LIN {X 0,Y 397.084,Z 365.643,A -85,B 0,C 180,E1 -11317.084,E2 -11317.084} C_VEL
LIN {X 0,Y 397.13,Z 365.642,A -85,B 0,C 180,E1 -11320.352,E2 -11320.352} C_VEL
LIN {X 0,Y 397.112,Z 365.642,A -85,B 0,C 180,E1 -11323.551,E2 -11323.551} C_VEL
LIN {X 0,Y 397.214,Z 365.628,A -85,B 0,C 180,E1 -11326.702,E2 -11326.702} C_VEL
LIN {X 0,Y 397.199,Z 365.633,A -85,B 0,C 180,E1 -11329.809,E2 -11329.809} C_VEL
LIN {X 0,Y 397.278,Z 365.619,A -85,B 0,C 180,E1 -11332.887,E2 -11332.887} C_VEL
LIN {X 0,Y 397.217,Z 365.627,A -85,B 0,C 180,E1 -11334.925,E2 -11334.925} C_VEL
LIN {X 0,Y 397.424,Z 365.608,A -85,B 0,C 180,E1 -11337.973,E2 -11337.973} C_VEL
LIN {X 0,Y 397.302,Z 365.616,A -85,B 0,C 180,E1 -11341.014,E2 -11341.014} C_VEL
LIN {X 0,Y 397.305,Z 365.616,A -85,B 0,C 180,E1 -11343.042,E2 -11343.042} C_VEL
LIN {X 0,Y 397.284,Z 365.62,A -85,B 0,C 180,E1 -11346.498,E2 -11346.498} C_VEL
LIN {X 0,Y 397.214,Z 365.627,A -85,B 0,C 180,E1 -11349.163,E2 -11349.163} C_VEL
LIN {X 0,Y 397.2,Z 365.633,A -85,B 0,C 180,E1 -11352.259,E2 -11352.259} C_VEL
LIN {X 0,Y 397.11,Z 365.642,A -85,B 0,C 180,E1 -11355.395,E2 -11355.395} C_VEL
LIN {X 0,Y 397.137,Z 365.638,A -85,B 0,C 180,E1 -11358.575,E2 -11358.575} C_VEL
LIN {X 0,Y 397.081,Z 365.65,A -85,B 0,C 180,E1 -11361.82,E2 -11361.82} C_VEL
LIN {X 0,Y 397.09,Z 365.643,A -85,B 0,C 180,E1 -11365.137,E2 -11365.137} C_VEL
LIN {X 0,Y 397.051,Z 365.648,A -85,B 0,C 180,E1 -11368.55,E2 -11368.55} C_VEL
LIN {X 0,Y 397.071,Z 365.652,A -85,B 0,C 180,E1 -11371.838,E2 -11371.838} C_VEL
LIN {X 0,Y 397.113,Z 365.641,A -85,B 0,C 180,E1 -11374.495,E2 -11374.495} C_VEL
LIN {X 0,Y 397.079,Z 365.646,A -85,B 0,C 180,E1 -11378.278,E2 -11378.278} C_VEL
LIN {X 0,Y 397.042,Z 365.654,A -85,B 0,C 180,E1 -11381.978,E2 -11381.978} C_VEL
LIN {X 0,Y 397.076,Z 365.645,A -85,B 0,C 180,E1 -11385.071,E2 -11385.071} C_VEL
LIN {X 0,Y 397.044,Z 365.653,A -85,B 0,C 180,E1 -11388.025,E2 -11388.025} C_VEL
LIN {X 0,Y 397.083,Z 365.65,A -85,B 0,C 180,E1 -11391.725,E2 -11391.725} C_VEL
LIN {X 0,Y 397.114,Z 365.643,A -85,B 0,C 180,E1 -11395.508,E2 -11395.508} C_VEL
LIN {X 0,Y 397.073,Z 365.646,A -85,B 0,C 180,E1 -11399.119,E2 -11399.119} C_VEL
LIN {X 0,Y 397.059,Z 365.648,A -85,B 0,C 180,E1 -11402.253,E2 -11402.253} C_VEL
LIN {X 0,Y 397.1,Z 365.641,A -85,B 0,C 180,E1 -11404.867,E2 -11404.867} C_VEL
LIN {X 0,Y 397.093,Z 365.645,A -85,B 0,C 180,E1 -11408.183,E2 -11408.183} C_VEL
LIN {X 0,Y 397.156,Z 365.638,A -85,B 0,C 180,E1 -11411.428,E2 -11411.428} C_VEL
LIN {X 0,Y 397.178,Z 365.632,A -85,B 0,C 180,E1 -11414.61,E2 -11414.61} C_VEL
LIN {X 0,Y 397.219,Z 365.633,A -85,B 0,C 180,E1 -11417.744,E2 -11417.744} C_VEL
LIN {X 0,Y 397.235,Z 365.625,A -85,B 0,C 180,E1 -11420.839,E2 -11420.839} C_VEL
LIN {X 0,Y 397.323,Z 365.618,A -85,B 0,C 180,E1 -11423.909,E2 -11423.909} C_VEL
LIN {X 0,Y 397.442,Z 365.602,A -85,B 0,C 180,E1 -11427.975,E2 -11427.975} C_VEL
LIN {X 0,Y 397.322,Z 365.615,A -85,B 0,C 180,E1 -11431.015,E2 -11431.015} C_VEL
LIN {X 0,Y 397.328,Z 365.614,A -85,B 0,C 180,E1 -11433.043,E2 -11433.043} C_VEL
LIN {X 0,Y 397.333,Z 365.614,A -85,B 0,C 180,E1 -11436.094,E2 -11436.094} C_VEL
LIN {X 0,Y 397.24,Z 365.626,A -85,B 0,C 180,E1 -11439.164,E2 -11439.164} C_VEL
LIN {X 0,Y 397.224,Z 365.627,A -85,B 0,C 180,E1 -11442.259,E2 -11442.259} C_VEL
LIN {X 0,Y 397.131,Z 365.642,A -85,B 0,C 180,E1 -11445.395,E2 -11445.395} C_VEL
LIN {X 0,Y 397.12,Z 365.639,A -85,B 0,C 180,E1 -11448.577,E2 -11448.577} C_VEL
LIN {X 0,Y 397.109,Z 365.644,A -85,B 0,C 180,E1 -11451.88,E2 -11451.88} C_VEL
LIN {X 0,Y 397.102,Z 365.648,A -85,B 0,C 180,E1 -11455.496,E2 -11455.496} C_VEL
LIN {X 0,Y 397.085,Z 365.644,A -85,B 0,C 180,E1 -11456.293,E2 -11456.293} C_VEL
LIN {X 0,Y 396.392,Z 365.734,A -85,B 0,C 180,E1 -11457.139,E2 -11457.139} C_VEL
LIN {X 0,Y 393.539,Z 366.085,A -85,B 0,C 180,E1 -11458.516,E2 -11458.516} C_VEL
LIN {X 0,Y 391.138,Z 366.39,A -85,B 0,C 180,E1 -11459.629,E2 -11459.629} C_VEL
LIN {X 0,Y 390.104,Z 366.514,A -85,B 0,C 180,E1 -11460.488,E2 -11460.488} C_VEL
LIN {X 0,Y 390.017,Z 366.524,A -85,B 0,C 180,E1 -11460.78,E2 -11460.78} C_VEL
LIN {X 0,Y 390.075,Z 366.518,A -85,B 0,C 180,E1 -11464.025,E2 -11464.025} C_VEL
LIN {X 0,Y 390.047,Z 366.527,A -85,B 0,C 180,E1 -11467.551,E2 -11467.551} C_VEL
LIN {X 0,Y 390.097,Z 366.671,A -85,B 0,C 180,E1 -11470.511,E2 -11470.511} C_VEL
LIN {X 0,Y 391.931,Z 374.358,A -85,B 0,C 180,E1 -11472.219,E2 -11472.219} C_VEL
LIN {X 0,Y 403.461,Z 402.483,A -85,B 0,C 180,E1 -11473.65,E2 -11473.65} C_VEL
LIN {X 0,Y 404.025,Z 406.025,A -85,B 0,C 180,E1 -11473.768,E2 -11473.768} C_VEL
LIN {X 0,Y 400.287,Z 540.12,A -85,B 0,C 180,E1 -11476.553,E2 -11476.553} C_VEL
LIN {X 0,Y 399.564,Z 555.692,A -85,B 0,C 180,E1 -11477.075,E2 -11477.075} C_VEL
LIN {X 0,Y 398.659,Z 570.442,A -85,B 0,C 180,E1 -11477.769,E2 -11477.769} C_VEL
LIN {X 0,Y 397.612,Z 584.806,A -85,B 0,C 180,E1 -11478.652,E2 -11478.652} C_VEL
LIN {X 0,Y 396.39,Z 599.024,A -85,B 0,C 180,E1 -11479.753,E2 -11479.753} C_VEL
LIN {X 0,Y 395.115,Z 612.215,A -85,B 0,C 180,E1 -11481.007,E2 -11481.007} C_VEL
LIN {X 0,Y 393.964,Z 623.855,A -85,B 0,C 180,E1 -11482.338,E2 -11482.338} C_VEL
LIN {X 0,Y 392.765,Z 634.668,A -85,B 0,C 180,E1 -11483.808,E2 -11483.808} C_VEL
LIN {X 0,Y 391.766,Z 644.273,A -85,B 0,C 180,E1 -11485.361,E2 -11485.361} C_VEL
LIN {X 0,Y 390.903,Z 653.106,A -85,B 0,C 180,E1 -11487.053,E2 -11487.053} C_VEL
LIN {X 0,Y 390.19,Z 660.807,A -85,B 0,C 180,E1 -11488.812,E2 -11488.812} C_VEL
LIN {X 0,Y 389.548,Z 668.117,A -85,B 0,C 180,E1 -11490.848,E2 -11490.848} C_VEL
LIN {X 0,Y 389.195,Z 673.427,A -85,B 0,C 180,E1 -11492.687,E2 -11492.687} C_VEL
LIN {X 0,Y 388.857,Z 677.865,A -85,B 0,C 180,E1 -11494.648,E2 -11494.648} C_VEL
LIN {X 0,Y 388.62,Z 680.999,A -85,B 0,C 180,E1 -11496.555,E2 -11496.555} C_VEL
LIN {X 0,Y 388.505,Z 683.357,A -85,B 0,C 180,E1 -11498.789,E2 -11498.789} C_VEL
LIN {X 0,Y 388.534,Z 684.131,A -85,B 0,C 180,E1 -11500.155,E2 -11500.155} C_VEL
LIN {X 0,Y 388.487,Z 684.268,A -85,B 0,C 180,E1 -11502.089,E2 -11502.089} C_VEL
LIN {X 0,Y 388.561,Z 683.211,A -85,B 0,C 180,E1 -11504.257,E2 -11504.257} C_VEL
LIN {X 0,Y 388.735,Z 680.867,A -85,B 0,C 180,E1 -11506.406,E2 -11506.406} C_VEL
LIN {X 0,Y 389.087,Z 677.216,A -85,B 0,C 180,E1 -11508.539,E2 -11508.539} C_VEL
LIN {X 0,Y 389.498,Z 672.229,A -85,B 0,C 180,E1 -11510.654,E2 -11510.654} C_VEL
LIN {X 0,Y 390.195,Z 665.771,A -85,B 0,C 180,E1 -11512.757,E2 -11512.757} C_VEL
LIN {X 0,Y 391.109,Z 657.684,A -85,B 0,C 180,E1 -11514.845,E2 -11514.845} C_VEL
LIN {X 0,Y 392.155,Z 649.088,A -85,B 0,C 180,E1 -11516.661,E2 -11516.661} C_VEL
LIN {X 0,Y 393.348,Z 639.841,A -85,B 0,C 180,E1 -11518.297,E2 -11518.297} C_VEL
LIN {X 0,Y 394.597,Z 629.967,A -85,B 0,C 180,E1 -11519.775,E2 -11519.775} C_VEL
LIN {X 0,Y 396.078,Z 618.007,A -85,B 0,C 180,E1 -11521.271,E2 -11521.271} C_VEL
LIN {X 0,Y 397.545,Z 605.861,A -85,B 0,C 180,E1 -11522.533,E2 -11522.533} C_VEL
LIN {X 0,Y 398.909,Z 592.833,A -85,B 0,C 180,E1 -11523.661,E2 -11523.661} C_VEL
LIN {X 0,Y 400.34,Z 577.558,A -85,B 0,C 180,E1 -11524.72,E2 -11524.72} C_VEL
LIN {X 0,Y 401.564,Z 562.455,A -85,B 0,C 180,E1 -11525.523,E2 -11525.523} C_VEL
LIN {X 0,Y 402.471,Z 547.733,A -85,B 0,C 180,E1 -11526.108,E2 -11526.108} C_VEL
LIN {X 0,Y 403.157,Z 530.189,A -85,B 0,C 180,E1 -11526.575,E2 -11526.575} C_VEL
LIN {X 0,Y 406.498,Z 444.552,A -85,B 0,C 180,E1 -11528.504,E2 -11528.504} C_VEL
LIN {X 0,Y 408.126,Z 406.872,A -85,B 0,C 180,E1 -11529.384,E2 -11529.384} C_VEL
LIN {X 0,Y 403.125,Z 395.638,A -85,B 0,C 180,E1 -11530.22,E2 -11530.22} C_VEL
LIN {X 0,Y 397.176,Z 384.365,A -85,B 0,C 180,E1 -11531.224,E2 -11531.224} C_VEL
LIN {X 0,Y 393.435,Z 377.468,A -85,B 0,C 180,E1 -11531.907,E2 -11531.907} C_VEL
LIN {X 0,Y 390.859,Z 368.87,A -85,B 0,C 180,E1 -11534.58,E2 -11534.58} C_VEL
LIN {X 0,Y 390.151,Z 366.515,A -85,B 0,C 180,E1 -11535.408,E2 -11535.408} C_VEL
LIN {X 0,Y 390.107,Z 366.518,A -85,B 0,C 180,E1 -11538.922,E2 -11538.922} C_VEL
LIN {X 0,Y 390.04,Z 366.527,A -85,B 0,C 180,E1 -11542.234,E2 -11542.234} C_VEL
LIN {X 0,Y 390.055,Z 366.523,A -85,B 0,C 180,E1 -11545.721,E2 -11545.721} C_VEL
LIN {X 0,Y 390.028,Z 366.527,A -85,B 0,C 180,E1 -11549.112,E2 -11549.112} C_VEL
LIN {X 0,Y 390.045,Z 366.523,A -85,B 0,C 180,E1 -11552.721,E2 -11552.721} C_VEL
LIN {X 0,Y 390.045,Z 366.524,A -85,B 0,C 180,E1 -11555.821,E2 -11555.821} C_VEL
LIN {X 0,Y 390.039,Z 366.523,A -85,B 0,C 180,E1 -11559.211,E2 -11559.211} C_VEL
LIN {X 0,Y 390.032,Z 366.525,A -85,B 0,C 180,E1 -11562.371,E2 -11562.371} C_VEL
LIN {X 0,Y 390.043,Z 366.522,A -85,B 0,C 180,E1 -11565.353,E2 -11565.353} C_VEL
LIN {X 0,Y 390.017,Z 366.529,A -85,B 0,C 180,E1 -11568.183,E2 -11568.183} C_VEL
LIN {X 0,Y 390.057,Z 366.524,A -85,B 0,C 180,E1 -11570.902,E2 -11570.902} C_VEL
LIN {X 0,Y 390.049,Z 366.622,A -85,B 0,C 180,E1 -11572.569,E2 -11572.569} C_VEL
LIN {X 0,Y 392.971,Z 375.911,A -85,B 0,C 180,E1 -11575.353,E2 -11575.353} C_VEL
LIN {X 0,Y 395.576,Z 385.111,A -85,B 0,C 180,E1 -11577.791,E2 -11577.791} C_VEL
LIN {X 0,Y 397.36,Z 392.743,A -85,B 0,C 180,E1 -11579.606,E2 -11579.606} C_VEL
LIN {X 0,Y 402.067,Z 403.196,A -85,B 0,C 180,E1 -11580.441,E2 -11580.441} C_VEL
LIN {X 0,Y 405.526,Z 420.641,A -85,B 0,C 180,E1 -11581.3,E2 -11581.3} C_VEL
LIN {X 0,Y 407.342,Z 433.31,A -85,B 0,C 180,E1 -11581.821,E2 -11581.821} C_VEL
LIN {X 0,Y 403.376,Z 535.394,A -85,B 0,C 180,E1 -11584.142,E2 -11584.142} C_VEL
LIN {X 0,Y 402.33,Z 562.211,A -85,B 0,C 180,E1 -11584.764,E2 -11584.764} C_VEL
LIN {X 0,Y 401.282,Z 577.923,A -85,B 0,C 180,E1 -11585.316,E2 -11585.316} C_VEL
LIN {X 0,Y 400.127,Z 591.639,A -85,B 0,C 180,E1 -11585.972,E2 -11585.972} C_VEL
LIN {X 0,Y 398.855,Z 605.345,A -85,B 0,C 180,E1 -11586.815,E2 -11586.815} C_VEL
LIN {X 0,Y 397.352,Z 619.705,A -85,B 0,C 180,E1 -11587.922,E2 -11587.922} C_VEL
LIN {X 0,Y 395.777,Z 633.199,A -85,B 0,C 180,E1 -11589.196,E2 -11589.196} C_VEL
LIN {X 0,Y 394.419,Z 644.547,A -85,B 0,C 180,E1 -11590.481,E2 -11590.481} C_VEL
LIN {X 0,Y 393.235,Z 654.197,A -85,B 0,C 180,E1 -11591.773,E2 -11591.773} C_VEL
LIN {X 0,Y 391.992,Z 664.177,A -85,B 0,C 180,E1 -11593.328,E2 -11593.328} C_VEL
LIN {X 0,Y 390.893,Z 673.993,A -85,B 0,C 180,E1 -11595.154,E2 -11595.154} C_VEL
LIN {X 0,Y 390.042,Z 682.44,A -85,B 0,C 180,E1 -11597.047,E2 -11597.047} C_VEL
LIN {X 0,Y 389.413,Z 689.832,A -85,B 0,C 180,E1 -11599.075,E2 -11599.075} C_VEL
LIN {X 0,Y 388.981,Z 695.897,A -85,B 0,C 180,E1 -11601.164,E2 -11601.164} C_VEL
LIN {X 0,Y 388.82,Z 699.512,A -85,B 0,C 180,E1 -11602.73,E2 -11602.73} C_VEL
LIN {X 0,Y 388.663,Z 703.134,A -85,B 0,C 180,E1 -11604.811,E2 -11604.811} C_VEL
LIN {X 0,Y 388.613,Z 705.481,A -85,B 0,C 180,E1 -11606.888,E2 -11606.888} C_VEL
LIN {X 0,Y 388.703,Z 706.605,A -85,B 0,C 180,E1 -11608.962,E2 -11608.962} C_VEL
LIN {X 0,Y 388.722,Z 706.513,A -85,B 0,C 180,E1 -11611.034,E2 -11611.034} C_VEL
LIN {X 0,Y 388.625,Z 705.186,A -85,B 0,C 180,E1 -11613.108,E2 -11613.108} C_VEL
LIN {X 0,Y 388.676,Z 702.579,A -85,B 0,C 180,E1 -11615.186,E2 -11615.186} C_VEL
LIN {X 0,Y 388.826,Z 698.67,A -85,B 0,C 180,E1 -11617.267,E2 -11617.267} C_VEL
LIN {X 0,Y 389.027,Z 693.361,A -85,B 0,C 180,E1 -11619.356,E2 -11619.356} C_VEL
LIN {X 0,Y 389.54,Z 686.524,A -85,B 0,C 180,E1 -11621.445,E2 -11621.445} C_VEL
LIN {X 0,Y 390.069,Z 678.742,A -85,B 0,C 180,E1 -11623.362,E2 -11623.362} C_VEL
LIN {X 0,Y 390.913,Z 670.161,A -85,B 0,C 180,E1 -11625.109,E2 -11625.109} C_VEL
LIN {X 0,Y 392.025,Z 659.37,A -85,B 0,C 180,E1 -11626.935,E2 -11626.935} C_VEL
LIN {X 0,Y 393.22,Z 647.776,A -85,B 0,C 180,E1 -11628.561,E2 -11628.561} C_VEL
LIN {X 0,Y 394.487,Z 634.924,A -85,B 0,C 180,E1 -11630.055,E2 -11630.055} C_VEL
LIN {X 0,Y 395.74,Z 622.851,A -85,B 0,C 180,E1 -11631.212,E2 -11631.212} C_VEL
LIN {X 0,Y 396.879,Z 609.966,A -85,B 0,C 180,E1 -11632.24,E2 -11632.24} C_VEL
LIN {X 0,Y 398.161,Z 595.409,A -85,B 0,C 180,E1 -11633.169,E2 -11633.169} C_VEL
LIN {X 0,Y 399.145,Z 580.132,A -85,B 0,C 180,E1 -11633.922,E2 -11633.922} C_VEL
LIN {X 0,Y 399.979,Z 565.003,A -85,B 0,C 180,E1 -11634.455,E2 -11634.455} C_VEL
LIN {X 0,Y 400.712,Z 542.464,A -85,B 0,C 180,E1 -11634.961,E2 -11634.961} C_VEL
LIN {X 0,Y 403.694,Z 431.306,A -85,B 0,C 180,E1 -11637.258,E2 -11637.258} C_VEL
LIN {X 0,Y 396.926,Z 395.43,A -85,B 0,C 180,E1 -11638.53,E2 -11638.53} C_VEL
LIN {X 0,Y 394.719,Z 385.401,A -85,B 0,C 180,E1 -11640.492,E2 -11640.492} C_VEL
LIN {X 0,Y 391.094,Z 370.654,A -85,B 0,C 180,E1 -11643.542,E2 -11643.542} C_VEL
LIN {X 0,Y 390.08,Z 366.52,A -85,B 0,C 180,E1 -11644.458,E2 -11644.458} C_VEL
LIN {X 0,Y 390.026,Z 366.528,A -85,B 0,C 180,E1 -11647.779,E2 -11647.779} C_VEL
LIN {X 0,Y 390.007,Z 366.526,A -85,B 0,C 180,E1 -11650.813,E2 -11650.813} C_VEL
LIN {X 0,Y 390.041,Z 366.524,A -85,B 0,C 180,E1 -11653.884,E2 -11653.884} C_VEL
LIN {X 0,Y 390.039,Z 366.522,A -85,B 0,C 180,E1 -11656.787,E2 -11656.787} C_VEL
LIN {X 0,Y 389.997,Z 366.527,A -85,B 0,C 180,E1 -11659.553,E2 -11659.553} C_VEL
LIN {X 0,Y 390.025,Z 366.527,A -85,B 0,C 180,E1 -11662.449,E2 -11662.449} C_VEL
LIN {X 0,Y 390.055,Z 366.525,A -85,B 0,C 180,E1 -11666.044,E2 -11666.044} C_VEL
LIN {X 0,Y 390.03,Z 366.526,A -85,B 0,C 180,E1 -11669.869,E2 -11669.869} C_VEL
LIN {X 0,Y 390.016,Z 366.524,A -85,B 0,C 180,E1 -11673.225,E2 -11673.225} C_VEL
LIN {X 0,Y 390.05,Z 366.52,A -85,B 0,C 180,E1 -11676.764,E2 -11676.764} C_VEL
LIN {X 0,Y 390.088,Z 366.521,A -85,B 0,C 180,E1 -11679.982,E2 -11679.982} C_VEL
LIN {X 0,Y 390.091,Z 366.515,A -85,B 0,C 180,E1 -11683.246,E2 -11683.246} C_VEL
LIN {X 0,Y 390.18,Z 366.505,A -85,B 0,C 180,E1 -11686.561,E2 -11686.561} C_VEL
LIN {X 0,Y 390.15,Z 366.51,A -85,B 0,C 180,E1 -11689.623,E2 -11689.623} C_VEL
LIN {X 0,Y 390.231,Z 366.498,A -85,B 0,C 180,E1 -11692.758,E2 -11692.758} C_VEL
LIN {X 0,Y 390.189,Z 366.503,A -85,B 0,C 180,E1 -11694.833,E2 -11694.833} C_VEL
LIN {X 0,Y 390.391,Z 366.483,A -85,B 0,C 180,E1 -11697.937,E2 -11697.937} C_VEL
LIN {X 0,Y 390.273,Z 366.492,A -85,B 0,C 180,E1 -11701.032,E2 -11701.032} C_VEL
LIN {X 0,Y 390.241,Z 366.496,A -85,B 0,C 180,E1 -11703.097,E2 -11703.097} C_VEL
LIN {X 0,Y 390.244,Z 366.497,A -85,B 0,C 180,E1 -11706.489,E2 -11706.489} C_VEL
LIN {X 0,Y 390.172,Z 366.505,A -85,B 0,C 180,E1 -11709.33,E2 -11709.33} C_VEL
LIN {X 0,Y 390.181,Z 366.505,A -85,B 0,C 180,E1 -11713.439,E2 -11713.439} C_VEL
LIN {X 0,Y 390.094,Z 366.515,A -85,B 0,C 180,E1 -11717.289,E2 -11717.289} C_VEL
LIN {X 0,Y 390.075,Z 366.518,A -85,B 0,C 180,E1 -11720.471,E2 -11720.471} C_VEL
LIN {X 0,Y 390.048,Z 366.521,A -85,B 0,C 180,E1 -11723.354,E2 -11723.354} C_VEL
LIN {X 0,Y 390.017,Z 366.524,A -85,B 0,C 180,E1 -11726.776,E2 -11726.776} C_VEL
LIN {X 0,Y 390.025,Z 366.525,A -85,B 0,C 180,E1 -11730.301,E2 -11730.301} C_VEL
LIN {X 0,Y 390.058,Z 366.524,A -85,B 0,C 180,E1 -11734.026,E2 -11734.026} C_VEL
LIN {X 0,Y 390.027,Z 366.526,A -85,B 0,C 180,E1 -11737.551,E2 -11737.551} C_VEL
LIN {X 0,Y 390.006,Z 366.525,A -85,B 0,C 180,E1 -11740.816,E2 -11740.816} C_VEL
LIN {X 0,Y 390.042,Z 366.527,A -85,B 0,C 180,E1 -11743.887,E2 -11743.887} C_VEL
LIN {X 0,Y 390.039,Z 366.521,A -85,B 0,C 180,E1 -11746.79,E2 -11746.79} C_VEL
LIN {X 0,Y 390.002,Z 366.53,A -85,B 0,C 180,E1 -11749.556,E2 -11749.556} C_VEL
LIN {X 0,Y 390.031,Z 366.523,A -85,B 0,C 180,E1 -11752.452,E2 -11752.452} C_VEL
LIN {X 0,Y 390.059,Z 366.522,A -85,B 0,C 180,E1 -11756.047,E2 -11756.047} C_VEL
LIN {X 0,Y 390.039,Z 366.527,A -85,B 0,C 180,E1 -11759.872,E2 -11759.872} C_VEL
LIN {X 0,Y 390.028,Z 366.524,A -85,B 0,C 180,E1 -11763.228,E2 -11763.228} C_VEL
LIN {X 0,Y 390.062,Z 366.518,A -85,B 0,C 180,E1 -11766.767,E2 -11766.767} C_VEL
LIN {X 0,Y 390.102,Z 366.517,A -85,B 0,C 180,E1 -11769.985,E2 -11769.985} C_VEL
LIN {X 0,Y 390.138,Z 366.511,A -85,B 0,C 180,E1 -11773.25,E2 -11773.25} C_VEL
LIN {X 0,Y 390.195,Z 366.502,A -85,B 0,C 180,E1 -11776.563,E2 -11776.563} C_VEL
LIN {X 0,Y 390.167,Z 366.511,A -85,B 0,C 180,E1 -11779.624,E2 -11779.624} C_VEL
LIN {X 0,Y 390.248,Z 366.495,A -85,B 0,C 180,E1 -11782.759,E2 -11782.759} C_VEL
LIN {X 0,Y 390.202,Z 366.501,A -85,B 0,C 180,E1 -11784.835,E2 -11784.835} C_VEL
LIN {X 0,Y 390.41,Z 366.479,A -85,B 0,C 180,E1 -11787.938,E2 -11787.938} C_VEL
LIN {X 0,Y 390.292,Z 366.49,A -85,B 0,C 180,E1 -11791.033,E2 -11791.033} C_VEL
LIN {X 0,Y 390.264,Z 366.494,A -85,B 0,C 180,E1 -11793.098,E2 -11793.098} C_VEL
LIN {X 0,Y 390.287,Z 366.491,A -85,B 0,C 180,E1 -11796.204,E2 -11796.204} C_VEL
LIN {X 0,Y 390.197,Z 366.505,A -85,B 0,C 180,E1 -11799.33,E2 -11799.33} C_VEL
LIN {X 0,Y 390.176,Z 366.504,A -85,B 0,C 180,E1 -11802.484,E2 -11802.484} C_VEL
LIN {X 0,Y 390.073,Z 366.523,A -85,B 0,C 180,E1 -11805.681,E2 -11805.681} C_VEL
LIN {X 0,Y 390.081,Z 366.517,A -85,B 0,C 180,E1 -11808.925,E2 -11808.925} C_VEL
LIN {X 0,Y 390.048,Z 366.521,A -85,B 0,C 180,E1 -11812.235,E2 -11812.235} C_VEL
LIN {X 0,Y 390.056,Z 366.524,A -85,B 0,C 180,E1 -11815.723,E2 -11815.723} C_VEL
LIN {X 0,Y 390.034,Z 366.524,A -85,B 0,C 180,E1 -11819.113,E2 -11819.113} C_VEL
LIN {X 0,Y 390.017,Z 366.524,A -85,B 0,C 180,E1 -11820.78,E2 -11820.78} C_VEL
LIN {X 0,Y 389.344,Z 366.613,A -85,B 0,C 180,E1 -11821.642,E2 -11821.642} C_VEL
LIN {X 0,Y 386.498,Z 366.964,A -85,B 0,C 180,E1 -11823.043,E2 -11823.043} C_VEL
LIN {X 0,Y 384.101,Z 367.262,A -85,B 0,C 180,E1 -11824.176,E2 -11824.176} C_VEL
LIN {X 0,Y 383.082,Z 367.39,A -85,B 0,C 180,E1 -11825.052,E2 -11825.052} C_VEL
LIN {X 0,Y 383.004,Z 367.398,A -85,B 0,C 180,E1 -11825.349,E2 -11825.349} C_VEL
LIN {X 0,Y 382.992,Z 367.404,A -85,B 0,C 180,E1 -11828.604,E2 -11828.604} C_VEL
LIN {X 0,Y 383.028,Z 367.544,A -85,B 0,C 180,E1 -11830.129,E2 -11830.129} C_VEL
LIN {X 0,Y 384.688,Z 374.387,A -85,B 0,C 180,E1 -11831.71,E2 -11831.71} C_VEL
LIN {X 0,Y 397.183,Z 404.809,A -85,B 0,C 180,E1 -11833.295,E2 -11833.295} C_VEL
LIN {X 0,Y 397.54,Z 406.565,A -85,B 0,C 180,E1 -11833.359,E2 -11833.359} C_VEL
LIN {X 0,Y 393.637,Z 540.349,A -85,B 0,C 180,E1 -11836.201,E2 -11836.201} C_VEL
LIN {X 0,Y 392.882,Z 555.985,A -85,B 0,C 180,E1 -11836.737,E2 -11836.737} C_VEL
LIN {X 0,Y 391.89,Z 571.329,A -85,B 0,C 180,E1 -11837.478,E2 -11837.478} C_VEL
LIN {X 0,Y 390.727,Z 586.229,A -85,B 0,C 180,E1 -11838.424,E2 -11838.424} C_VEL
LIN {X 0,Y 389.538,Z 599.69,A -85,B 0,C 180,E1 -11839.495,E2 -11839.495} C_VEL
LIN {X 0,Y 388.31,Z 612.109,A -85,B 0,C 180,E1 -11840.693,E2 -11840.693} C_VEL
LIN {X 0,Y 386.989,Z 624.954,A -85,B 0,C 180,E1 -11842.198,E2 -11842.198} C_VEL
LIN {X 0,Y 385.754,Z 635.657,A -85,B 0,C 180,E1 -11843.692,E2 -11843.692} C_VEL
LIN {X 0,Y 384.637,Z 646.401,A -85,B 0,C 180,E1 -11845.498,E2 -11845.498} C_VEL
LIN {X 0,Y 383.65,Z 655.865,A -85,B 0,C 180,E1 -11847.424,E2 -11847.424} C_VEL
LIN {X 0,Y 382.891,Z 663.855,A -85,B 0,C 180,E1 -11849.406,E2 -11849.406} C_VEL
LIN {X 0,Y 382.343,Z 670.525,A -85,B 0,C 180,E1 -11851.45,E2 -11851.45} C_VEL
LIN {X 0,Y 381.996,Z 675.112,A -85,B 0,C 180,E1 -11853.208,E2 -11853.208} C_VEL
LIN {X 0,Y 381.696,Z 678.692,A -85,B 0,C 180,E1 -11854.945,E2 -11854.945} C_VEL
LIN {X 0,Y 381.486,Z 682.083,A -85,B 0,C 180,E1 -11857.239,E2 -11857.239} C_VEL
LIN {X 0,Y 381.413,Z 684.001,A -85,B 0,C 180,E1 -11859.506,E2 -11859.506} C_VEL
LIN {X 0,Y 381.407,Z 684.535,A -85,B 0,C 180,E1 -11861.744,E2 -11861.744} C_VEL
LIN {X 0,Y 381.463,Z 683.742,A -85,B 0,C 180,E1 -11863.957,E2 -11863.957} C_VEL
LIN {X 0,Y 381.607,Z 681.66,A -85,B 0,C 180,E1 -11866.147,E2 -11866.147} C_VEL
LIN {X 0,Y 381.994,Z 678.261,A -85,B 0,C 180,E1 -11868.323,E2 -11868.323} C_VEL
LIN {X 0,Y 382.413,Z 673.529,A -85,B 0,C 180,E1 -11870.479,E2 -11870.479} C_VEL
LIN {X 0,Y 383.102,Z 667.352,A -85,B 0,C 180,E1 -11872.622,E2 -11872.622} C_VEL
LIN {X 0,Y 384.059,Z 659.606,A -85,B 0,C 180,E1 -11874.75,E2 -11874.75} C_VEL
LIN {X 0,Y 385.101,Z 651.364,A -85,B 0,C 180,E1 -11876.599,E2 -11876.599} C_VEL
LIN {X 0,Y 386.474,Z 641.139,A -85,B 0,C 180,E1 -11878.489,E2 -11878.489} C_VEL
LIN {X 0,Y 387.78,Z 631.338,A -85,B 0,C 180,E1 -11880,E2 -11880} C_VEL
LIN {X 0,Y 389.368,Z 619.381,A -85,B 0,C 180,E1 -11881.551,E2 -11881.551} C_VEL
LIN {X 0,Y 391.073,Z 606.192,A -85,B 0,C 180,E1 -11882.961,E2 -11882.961} C_VEL
LIN {X 0,Y 392.503,Z 593.192,A -85,B 0,C 180,E1 -11884.107,E2 -11884.107} C_VEL
LIN {X 0,Y 394.018,Z 577.93,A -85,B 0,C 180,E1 -11885.181,E2 -11885.181} C_VEL
LIN {X 0,Y 395.309,Z 562.852,A -85,B 0,C 180,E1 -11885.995,E2 -11885.995} C_VEL
LIN {X 0,Y 396.251,Z 548.202,A -85,B 0,C 180,E1 -11886.594,E2 -11886.594} C_VEL
LIN {X 0,Y 396.992,Z 531.621,A -85,B 0,C 180,E1 -11887.054,E2 -11887.054} C_VEL
LIN {X 0,Y 400.572,Z 445.139,A -85,B 0,C 180,E1 -11889.051,E2 -11889.051} C_VEL
LIN {X 0,Y 402.229,Z 409.013,A -85,B 0,C 180,E1 -11889.926,E2 -11889.926} C_VEL
LIN {X 0,Y 397.462,Z 398.428,A -85,B 0,C 180,E1 -11890.754,E2 -11890.754} C_VEL
LIN {X 0,Y 392.158,Z 388.24,A -85,B 0,C 180,E1 -11891.703,E2 -11891.703} C_VEL
LIN {X 0,Y 386.355,Z 377.892,A -85,B 0,C 180,E1 -11892.808,E2 -11892.808} C_VEL
LIN {X 0,Y 383.94,Z 370.084,A -85,B 0,C 180,E1 -11895.392,E2 -11895.392} C_VEL
LIN {X 0,Y 383.084,Z 367.396,A -85,B 0,C 180,E1 -11896.383,E2 -11896.383} C_VEL
LIN {X 0,Y 383.064,Z 367.396,A -85,B 0,C 180,E1 -11899.283,E2 -11899.283} C_VEL
LIN {X 0,Y 382.993,Z 367.403,A -85,B 0,C 180,E1 -11902.665,E2 -11902.665} C_VEL
LIN {X 0,Y 382.987,Z 367.406,A -85,B 0,C 180,E1 -11906.13,E2 -11906.13} C_VEL
LIN {X 0,Y 382.979,Z 367.404,A -85,B 0,C 180,E1 -11909.701,E2 -11909.701} C_VEL
LIN {X 0,Y 383.003,Z 367.401,A -85,B 0,C 180,E1 -11913.4,E2 -11913.4} C_VEL
LIN {X 0,Y 383.025,Z 367.399,A -85,B 0,C 180,E1 -11916.161,E2 -11916.161} C_VEL
LIN {X 0,Y 382.988,Z 367.403,A -85,B 0,C 180,E1 -11919.58,E2 -11919.58} C_VEL
LIN {X 0,Y 383.01,Z 367.4,A -85,B 0,C 180,E1 -11922.778,E2 -11922.778} C_VEL
LIN {X 0,Y 382.992,Z 367.402,A -85,B 0,C 180,E1 -11925.787,E2 -11925.787} C_VEL
LIN {X 0,Y 382.964,Z 367.404,A -85,B 0,C 180,E1 -11928.8,E2 -11928.8} C_VEL
LIN {X 0,Y 382.994,Z 367.542,A -85,B 0,C 180,E1 -11931.595,E2 -11931.595} C_VEL
LIN {X 0,Y 386.101,Z 377.031,A -85,B 0,C 180,E1 -11934.64,E2 -11934.64} C_VEL
LIN {X 0,Y 388.639,Z 386.04,A -85,B 0,C 180,E1 -11937.144,E2 -11937.144} C_VEL
LIN {X 0,Y 390.203,Z 392.381,A -85,B 0,C 180,E1 -11938.736,E2 -11938.736} C_VEL
LIN {X 0,Y 396.709,Z 406.322,A -85,B 0,C 180,E1 -11939.949,E2 -11939.949} C_VEL
LIN {X 0,Y 400.181,Z 424.732,A -85,B 0,C 180,E1 -11940.868,E2 -11940.868} C_VEL
LIN {X 0,Y 401.454,Z 433.668,A -85,B 0,C 180,E1 -11941.259,E2 -11941.259} C_VEL
LIN {X 0,Y 397.172,Z 537.219,A -85,B 0,C 180,E1 -11943.672,E2 -11943.672} C_VEL
LIN {X 0,Y 396.044,Z 562.963,A -85,B 0,C 180,E1 -11944.299,E2 -11944.299} C_VEL
LIN {X 0,Y 394.861,Z 579.409,A -85,B 0,C 180,E1 -11944.904,E2 -11944.904} C_VEL
LIN {X 0,Y 393.586,Z 593.649,A -85,B 0,C 180,E1 -11945.625,E2 -11945.625} C_VEL
LIN {X 0,Y 392.147,Z 607.597,A -85,B 0,C 180,E1 -11946.529,E2 -11946.529} C_VEL
LIN {X 0,Y 390.591,Z 621.52,A -85,B 0,C 180,E1 -11947.658,E2 -11947.658} C_VEL
LIN {X 0,Y 388.988,Z 634.598,A -85,B 0,C 180,E1 -11948.954,E2 -11948.954} C_VEL
LIN {X 0,Y 387.436,Z 646.678,A -85,B 0,C 180,E1 -11950.391,E2 -11950.391} C_VEL
LIN {X 0,Y 386.229,Z 656.237,A -85,B 0,C 180,E1 -11951.723,E2 -11951.723} C_VEL
LIN {X 0,Y 384.806,Z 667.247,A -85,B 0,C 180,E1 -11953.554,E2 -11953.554} C_VEL
LIN {X 0,Y 383.678,Z 676.519,A -85,B 0,C 180,E1 -11955.411,E2 -11955.411} C_VEL
LIN {X 0,Y 382.861,Z 684.234,A -85,B 0,C 180,E1 -11957.273,E2 -11957.273} C_VEL
LIN {X 0,Y 382.391,Z 689.753,A -85,B 0,C 180,E1 -11958.872,E2 -11958.872} C_VEL
LIN {X 0,Y 381.904,Z 695.788,A -85,B 0,C 180,E1 -11960.999,E2 -11960.999} C_VEL
LIN {X 0,Y 381.729,Z 699.392,A -85,B 0,C 180,E1 -11962.594,E2 -11962.594} C_VEL
LIN {X 0,Y 381.575,Z 702.987,A -85,B 0,C 180,E1 -11964.715,E2 -11964.715} C_VEL
LIN {X 0,Y 381.523,Z 705.307,A -85,B 0,C 180,E1 -11966.831,E2 -11966.831} C_VEL
LIN {X 0,Y 381.617,Z 706.402,A -85,B 0,C 180,E1 -11968.943,E2 -11968.943} C_VEL
LIN {X 0,Y 381.636,Z 706.277,A -85,B 0,C 180,E1 -11971.054,E2 -11971.054} C_VEL
LIN {X 0,Y 381.536,Z 704.918,A -85,B 0,C 180,E1 -11973.166,E2 -11973.166} C_VEL
LIN {X 0,Y 381.584,Z 702.281,A -85,B 0,C 180,E1 -11975.282,E2 -11975.282} C_VEL
LIN {X 0,Y 381.732,Z 698.324,A -85,B 0,C 180,E1 -11977.403,E2 -11977.403} C_VEL
LIN {X 0,Y 381.968,Z 692.959,A -85,B 0,C 180,E1 -11979.53,E2 -11979.53} C_VEL
LIN {X 0,Y 382.509,Z 686.057,A -85,B 0,C 180,E1 -11981.658,E2 -11981.658} C_VEL
LIN {X 0,Y 383.03,Z 678.78,A -85,B 0,C 180,E1 -11983.477,E2 -11983.477} C_VEL
LIN {X 0,Y 383.948,Z 669.542,A -85,B 0,C 180,E1 -11985.39,E2 -11985.39} C_VEL
LIN {X 0,Y 384.939,Z 660.332,A -85,B 0,C 180,E1 -11986.983,E2 -11986.983} C_VEL
LIN {X 0,Y 386.169,Z 649.054,A -85,B 0,C 180,E1 -11988.624,E2 -11988.624} C_VEL
LIN {X 0,Y 387.459,Z 636.368,A -85,B 0,C 180,E1 -11990.158,E2 -11990.158} C_VEL
LIN {X 0,Y 388.878,Z 623.188,A -85,B 0,C 180,E1 -11991.465,E2 -11991.465} C_VEL
LIN {X 0,Y 390.057,Z 610.418,A -85,B 0,C 180,E1 -11992.51,E2 -11992.51} C_VEL
LIN {X 0,Y 391.403,Z 595.814,A -85,B 0,C 180,E1 -11993.466,E2 -11993.466} C_VEL
LIN {X 0,Y 392.437,Z 580.365,A -85,B 0,C 180,E1 -11994.249,E2 -11994.249} C_VEL
LIN {X 0,Y 393.299,Z 565.385,A -85,B 0,C 180,E1 -11994.793,E2 -11994.793} C_VEL
LIN {X 0,Y 394.048,Z 544.903,A -85,B 0,C 180,E1 -11995.271,E2 -11995.271} C_VEL
LIN {X 0,Y 397.188,Z 432.389,A -85,B 0,C 180,E1 -11997.647,E2 -11997.647} C_VEL
LIN {X 0,Y 390.796,Z 398.106,A -85,B 0,C 180,E1 -11998.885,E2 -11998.885} C_VEL
LIN {X 0,Y 389.681,Z 394.961,A -85,B 0,C 180,E1 -11999.064,E2 -11999.064} C_VEL
LIN {X 0,Y 386.171,Z 379.966,A -85,B 0,C 180,E1 -12002.134,E2 -12002.134} C_VEL
LIN {X 0,Y 383.046,Z 367.395,A -85,B 0,C 180,E1 -12004.863,E2 -12004.863} C_VEL
LIN {X 0,Y 382.971,Z 367.407,A -85,B 0,C 180,E1 -12008.602,E2 -12008.602} C_VEL
LIN {X 0,Y 382.95,Z 367.404,A -85,B 0,C 180,E1 -12011.349,E2 -12011.349} C_VEL
LIN {X 0,Y 382.983,Z 367.406,A -85,B 0,C 180,E1 -12014.302,E2 -12014.302} C_VEL
LIN {X 0,Y 382.999,Z 367.398,A -85,B 0,C 180,E1 -12017.239,E2 -12017.239} C_VEL
LIN {X 0,Y 382.972,Z 367.405,A -85,B 0,C 180,E1 -12020.418,E2 -12020.418} C_VEL
LIN {X 0,Y 383.004,Z 367.403,A -85,B 0,C 180,E1 -12024.042,E2 -12024.042} C_VEL
LIN {X 0,Y 382.974,Z 367.403,A -85,B 0,C 180,E1 -12027.577,E2 -12027.577} C_VEL
LIN {X 0,Y 382.962,Z 367.407,A -85,B 0,C 180,E1 -12030.298,E2 -12030.298} C_VEL
LIN {X 0,Y 382.988,Z 367.406,A -85,B 0,C 180,E1 -12034.044,E2 -12034.044} C_VEL
LIN {X 0,Y 382.974,Z 367.402,A -85,B 0,C 180,E1 -12037.333,E2 -12037.333} C_VEL
LIN {X 0,Y 383.041,Z 367.394,A -85,B 0,C 180,E1 -12040.716,E2 -12040.716} C_VEL
LIN {X 0,Y 383.005,Z 367.404,A -85,B 0,C 180,E1 -12044.024,E2 -12044.024} C_VEL
LIN {X 0,Y 383.121,Z 367.383,A -85,B 0,C 180,E1 -12047.284,E2 -12047.284} C_VEL
LIN {X 0,Y 383.127,Z 367.384,A -85,B 0,C 180,E1 -12050.498,E2 -12050.498} C_VEL
LIN {X 0,Y 383.224,Z 367.373,A -85,B 0,C 180,E1 -12053.683,E2 -12053.683} C_VEL
LIN {X 0,Y 383.357,Z 367.359,A -85,B 0,C 180,E1 -12057.899,E2 -12057.899} C_VEL
LIN {X 0,Y 383.244,Z 367.367,A -85,B 0,C 180,E1 -12061.051,E2 -12061.051} C_VEL
LIN {X 0,Y 383.357,Z 367.359,A -85,B 0,C 180,E1 -12062.102,E2 -12062.102} C_VEL
LIN {X 0,Y 383.209,Z 367.374,A -85,B 0,C 180,E1 -12066.476,E2 -12066.476} C_VEL
LIN {X 0,Y 383.123,Z 367.385,A -85,B 0,C 180,E1 -12069.503,E2 -12069.503} C_VEL
LIN {X 0,Y 383.112,Z 367.386,A -85,B 0,C 180,E1 -12073.537,E2 -12073.537} C_VEL
LIN {X 0,Y 383.044,Z 367.394,A -85,B 0,C 180,E1 -12077.438,E2 -12077.438} C_VEL
LIN {X 0,Y 383.016,Z 367.396,A -85,B 0,C 180,E1 -12080.648,E2 -12080.648} C_VEL
LIN {X 0,Y 382.997,Z 367.404,A -85,B 0,C 180,E1 -12083.81,E2 -12083.81} C_VEL
LIN {X 0,Y 382.957,Z 367.404,A -85,B 0,C 180,E1 -12087.31,E2 -12087.31} C_VEL
LIN {X 0,Y 382.97,Z 367.402,A -85,B 0,C 180,E1 -12090.92,E2 -12090.92} C_VEL
LIN {X 0,Y 383.003,Z 367.398,A -85,B 0,C 180,E1 -12094.67,E2 -12094.67} C_VEL
LIN {X 0,Y 382.982,Z 367.407,A -85,B 0,C 180,E1 -12097.904,E2 -12097.904} C_VEL
LIN {X 0,Y 382.951,Z 367.406,A -85,B 0,C 180,E1 -12101.352,E2 -12101.352} C_VEL
LIN {X 0,Y 382.984,Z 367.402,A -85,B 0,C 180,E1 -12104.304,E2 -12104.304} C_VEL
LIN {X 0,Y 382.988,Z 367.401,A -85,B 0,C 180,E1 -12107.24,E2 -12107.24} C_VEL
LIN {X 0,Y 382.978,Z 367.402,A -85,B 0,C 180,E1 -12110.421,E2 -12110.421} C_VEL
LIN {X 0,Y 383.008,Z 367.401,A -85,B 0,C 180,E1 -12114.045,E2 -12114.045} C_VEL
LIN {X 0,Y 382.981,Z 367.405,A -85,B 0,C 180,E1 -12117.58,E2 -12117.58} C_VEL
LIN {X 0,Y 382.972,Z 367.403,A -85,B 0,C 180,E1 -12120.301,E2 -12120.301} C_VEL
LIN {X 0,Y 382.999,Z 367.402,A -85,B 0,C 180,E1 -12124.047,E2 -12124.047} C_VEL
LIN {X 0,Y 382.986,Z 367.402,A -85,B 0,C 180,E1 -12127.336,E2 -12127.336} C_VEL
LIN {X 0,Y 383.057,Z 367.391,A -85,B 0,C 180,E1 -12130.718,E2 -12130.718} C_VEL
LIN {X 0,Y 383.08,Z 367.391,A -85,B 0,C 180,E1 -12134.028,E2 -12134.028} C_VEL
LIN {X 0,Y 383.137,Z 367.383,A -85,B 0,C 180,E1 -12137.286,E2 -12137.286} C_VEL
LIN {X 0,Y 383.143,Z 367.38,A -85,B 0,C 180,E1 -12140.499,E2 -12140.499} C_VEL
LIN {X 0,Y 383.236,Z 367.376,A -85,B 0,C 180,E1 -12143.685,E2 -12143.685} C_VEL
LIN {X 0,Y 383.376,Z 367.355,A -85,B 0,C 180,E1 -12147.9,E2 -12147.9} C_VEL
LIN {X 0,Y 383.263,Z 367.366,A -85,B 0,C 180,E1 -12151.052,E2 -12151.052} C_VEL
LIN {X 0,Y 383.377,Z 367.353,A -85,B 0,C 180,E1 -12152.103,E2 -12152.103} C_VEL
LIN {X 0,Y 383.244,Z 367.368,A -85,B 0,C 180,E1 -12156.318,E2 -12156.318} C_VEL
LIN {X 0,Y 383.148,Z 367.385,A -85,B 0,C 180,E1 -12159.504,E2 -12159.504} C_VEL
LIN {X 0,Y 383.131,Z 367.388,A -85,B 0,C 180,E1 -12163.537,E2 -12163.537} C_VEL
LIN {X 0,Y 383.06,Z 367.396,A -85,B 0,C 180,E1 -12167.436,E2 -12167.436} C_VEL
LIN {X 0,Y 383.037,Z 367.393,A -85,B 0,C 180,E1 -12170.649,E2 -12170.649} C_VEL
LIN {X 0,Y 383.015,Z 367.4,A -85,B 0,C 180,E1 -12173.81,E2 -12173.81} C_VEL
LIN {X 0,Y 382.987,Z 367.404,A -85,B 0,C 180,E1 -12177.309,E2 -12177.309} C_VEL
LIN {X 0,Y 382.989,Z 367.4,A -85,B 0,C 180,E1 -12180.919,E2 -12180.919} C_VEL
LIN {X 0,Y 383.025,Z 367.395,A -85,B 0,C 180,E1 -12184.669,E2 -12184.669} C_VEL
LIN {X 0,Y 383.004,Z 367.398,A -85,B 0,C 180,E1 -12185.349,E2 -12185.349} C_VEL
LIN {X 0,Y 382.336,Z 367.488,A -85,B 0,C 180,E1 -12185.934,E2 -12185.934} C_VEL
LIN {X 0,Y 379.501,Z 367.841,A -85,B 0,C 180,E1 -12186.85,E2 -12186.85} C_VEL
LIN {X 0,Y 376.633,Z 368.197,A -85,B 0,C 180,E1 -12187.778,E2 -12187.778} C_VEL
LIN {X 0,Y 375.939,Z 368.28,A -85,B 0,C 180,E1 -12188.379,E2 -12188.379} C_VEL
LIN {X 0,Y 375.98,Z 368.361,A -85,B 0,C 180,E1 -12189.72,E2 -12189.72} C_VEL
LIN {X 0,Y 377.511,Z 374.712,A -85,B 0,C 180,E1 -12191.192,E2 -12191.192} C_VEL
LIN {X 0,Y 390.151,Z 405.216,A -85,B 0,C 180,E1 -12192.841,E2 -12192.841} C_VEL
LIN {X 0,Y 391.051,Z 407.757,A -85,B 0,C 180,E1 -12192.961,E2 -12192.961} C_VEL
LIN {X 0,Y 386.983,Z 540.399,A -85,B 0,C 180,E1 -12195.841,E2 -12195.841} C_VEL
LIN {X 0,Y 386.186,Z 556.145,A -85,B 0,C 180,E1 -12196.389,E2 -12196.389} C_VEL
LIN {X 0,Y 385.199,Z 571.353,A -85,B 0,C 180,E1 -12197.136,E2 -12197.136} C_VEL
LIN {X 0,Y 384.015,Z 586.13,A -85,B 0,C 180,E1 -12198.087,E2 -12198.087} C_VEL
LIN {X 0,Y 382.794,Z 599.382,A -85,B 0,C 180,E1 -12199.151,E2 -12199.151} C_VEL
LIN {X 0,Y 381.365,Z 613.209,A -85,B 0,C 180,E1 -12200.516,E2 -12200.516} C_VEL
LIN {X 0,Y 380.131,Z 624.804,A -85,B 0,C 180,E1 -12201.899,E2 -12201.899} C_VEL
LIN {X 0,Y 378.737,Z 636.521,A -85,B 0,C 180,E1 -12203.572,E2 -12203.572} C_VEL
LIN {X 0,Y 377.603,Z 647.166,A -85,B 0,C 180,E1 -12205.412,E2 -12205.412} C_VEL
LIN {X 0,Y 376.634,Z 655.974,A -85,B 0,C 180,E1 -12207.238,E2 -12207.238} C_VEL
LIN {X 0,Y 375.844,Z 664.271,A -85,B 0,C 180,E1 -12209.337,E2 -12209.337} C_VEL
LIN {X 0,Y 375.292,Z 670.658,A -85,B 0,C 180,E1 -12211.328,E2 -12211.328} C_VEL
LIN {X 0,Y 374.904,Z 675.604,A -85,B 0,C 180,E1 -12213.262,E2 -12213.262} C_VEL
LIN {X 0,Y 374.607,Z 679.106,A -85,B 0,C 180,E1 -12215.031,E2 -12215.031} C_VEL
LIN {X 0,Y 374.429,Z 681.899,A -85,B 0,C 180,E1 -12216.888,E2 -12216.888} C_VEL
LIN {X 0,Y 374.301,Z 683.983,A -85,B 0,C 180,E1 -12219.099,E2 -12219.099} C_VEL
LIN {X 0,Y 374.339,Z 684.554,A -85,B 0,C 180,E1 -12220.248,E2 -12220.248} C_VEL
LIN {X 0,Y 374.309,Z 684.668,A -85,B 0,C 180,E1 -12222.517,E2 -12222.517} C_VEL
LIN {X 0,Y 374.394,Z 683.459,A -85,B 0,C 180,E1 -12224.763,E2 -12224.763} C_VEL
LIN {X 0,Y 374.699,Z 680.598,A -85,B 0,C 180,E1 -12227.251,E2 -12227.251} C_VEL
LIN {X 0,Y 375.035,Z 677.138,A -85,B 0,C 180,E1 -12229.199,E2 -12229.199} C_VEL
LIN {X 0,Y 375.572,Z 671.988,A -85,B 0,C 180,E1 -12231.39,E2 -12231.39} C_VEL
LIN {X 0,Y 376.435,Z 665.355,A -85,B 0,C 180,E1 -12233.568,E2 -12233.568} C_VEL
LIN {X 0,Y 377.396,Z 658.201,A -85,B 0,C 180,E1 -12235.46,E2 -12235.46} C_VEL
LIN {X 0,Y 378.575,Z 649.609,A -85,B 0,C 180,E1 -12237.34,E2 -12237.34} C_VEL
LIN {X 0,Y 380.135,Z 639.143,A -85,B 0,C 180,E1 -12239.233,E2 -12239.233} C_VEL
LIN {X 0,Y 381.526,Z 628.868,A -85,B 0,C 180,E1 -12240.791,E2 -12240.791} C_VEL
LIN {X 0,Y 383.282,Z 616.344,A -85,B 0,C 180,E1 -12242.364,E2 -12242.364} C_VEL
LIN {X 0,Y 385.09,Z 602.434,A -85,B 0,C 180,E1 -12243.793,E2 -12243.793} C_VEL
LIN {X 0,Y 386.671,Z 588.584,A -85,B 0,C 180,E1 -12244.952,E2 -12244.952} C_VEL
LIN {X 0,Y 388.14,Z 574.24,A -85,B 0,C 180,E1 -12245.911,E2 -12245.911} C_VEL
LIN {X 0,Y 389.399,Z 558.967,A -85,B 0,C 180,E1 -12246.7,E2 -12246.7} C_VEL
LIN {X 0,Y 390.456,Z 542.96,A -85,B 0,C 180,E1 -12247.292,E2 -12247.292} C_VEL
LIN {X 0,Y 395.805,Z 424.812,A -85,B 0,C 180,E1 -12250.14,E2 -12250.14} C_VEL
LIN {X 0,Y 396.436,Z 411.164,A -85,B 0,C 180,E1 -12250.485,E2 -12250.485} C_VEL
LIN {X 0,Y 391.543,Z 400.404,A -85,B 0,C 180,E1 -12251.387,E2 -12251.387} C_VEL
LIN {X 0,Y 384.322,Z 386.872,A -85,B 0,C 180,E1 -12252.753,E2 -12252.753} C_VEL
LIN {X 0,Y 380.656,Z 380.963,A -85,B 0,C 180,E1 -12253.47,E2 -12253.47} C_VEL
LIN {X 0,Y 379.224,Z 378.313,A -85,B 0,C 180,E1 -12253.804,E2 -12253.804} C_VEL
LIN {X 0,Y 377.035,Z 371.453,A -85,B 0,C 180,E1 -12256.236,E2 -12256.236} C_VEL
LIN {X 0,Y 376.033,Z 368.274,A -85,B 0,C 180,E1 -12257.496,E2 -12257.496} C_VEL
LIN {X 0,Y 375.984,Z 368.278,A -85,B 0,C 180,E1 -12260.831,E2 -12260.831} C_VEL
LIN {X 0,Y 375.964,Z 368.279,A -85,B 0,C 180,E1 -12264.283,E2 -12264.283} C_VEL
LIN {X 0,Y 375.922,Z 368.285,A -85,B 0,C 180,E1 -12267.864,E2 -12267.864} C_VEL
LIN {X 0,Y 375.958,Z 368.28,A -85,B 0,C 180,E1 -12270.692,E2 -12270.692} C_VEL
LIN {X 0,Y 375.961,Z 368.279,A -85,B 0,C 180,E1 -12274.111,E2 -12274.111} C_VEL
LIN {X 0,Y 375.951,Z 368.281,A -85,B 0,C 180,E1 -12276.741,E2 -12276.741} C_VEL
LIN {X 0,Y 375.941,Z 368.282,A -85,B 0,C 180,E1 -12279.96,E2 -12279.96} C_VEL
LIN {X 0,Y 375.927,Z 368.281,A -85,B 0,C 180,E1 -12283.766,E2 -12283.766} C_VEL
LIN {X 0,Y 375.936,Z 368.281,A -85,B 0,C 180,E1 -12286.81,E2 -12286.81} C_VEL
LIN {X 0,Y 375.964,Z 368.318,A -85,B 0,C 180,E1 -12290.474,E2 -12290.474} C_VEL
LIN {X 0,Y 378.32,Z 375.549,A -85,B 0,C 180,E1 -12293.016,E2 -12293.016} C_VEL
LIN {X 0,Y 380.692,Z 383.229,A -85,B 0,C 180,E1 -12295.391,E2 -12295.391} C_VEL
LIN {X 0,Y 383.055,Z 392.047,A -85,B 0,C 180,E1 -12297.795,E2 -12297.795} C_VEL
LIN {X 0,Y 389.677,Z 405.53,A -85,B 0,C 180,E1 -12299.096,E2 -12299.096} C_VEL
LIN {X 0,Y 391.598,Z 410.38,A -85,B 0,C 180,E1 -12299.48,E2 -12299.48} C_VEL
LIN {X 0,Y 394.882,Z 428.859,A -85,B 0,C 180,E1 -12300.424,E2 -12300.424} C_VEL
LIN {X 0,Y 395.637,Z 435.429,A -85,B 0,C 180,E1 -12300.7,E2 -12300.7} C_VEL
LIN {X 0,Y 391.354,Z 531.071,A -85,B 0,C 180,E1 -12302.998,E2 -12302.998} C_VEL
LIN {X 0,Y 389.947,Z 562.318,A -85,B 0,C 180,E1 -12303.759,E2 -12303.759} C_VEL
LIN {X 0,Y 388.739,Z 578.342,A -85,B 0,C 180,E1 -12304.356,E2 -12304.356} C_VEL
LIN {X 0,Y 387.422,Z 592.148,A -85,B 0,C 180,E1 -12305.053,E2 -12305.053} C_VEL
LIN {X 0,Y 385.873,Z 606.746,A -85,B 0,C 180,E1 -12306.007,E2 -12306.007} C_VEL
LIN {X 0,Y 384.458,Z 619.1,A -85,B 0,C 180,E1 -12306.998,E2 -12306.998} C_VEL
LIN {X 0,Y 382.694,Z 632.56,A -85,B 0,C 180,E1 -12308.308,E2 -12308.308} C_VEL
LIN {X 0,Y 380.995,Z 644.908,A -85,B 0,C 180,E1 -12309.764,E2 -12309.764} C_VEL
LIN {X 0,Y 379.419,Z 656.488,A -85,B 0,C 180,E1 -12311.408,E2 -12311.408} C_VEL
LIN {X 0,Y 377.928,Z 667.287,A -85,B 0,C 180,E1 -12313.246,E2 -12313.246} C_VEL
LIN {X 0,Y 376.744,Z 676.529,A -85,B 0,C 180,E1 -12315.136,E2 -12315.136} C_VEL
LIN {X 0,Y 375.884,Z 684.231,A -85,B 0,C 180,E1 -12317.033,E2 -12317.033} C_VEL
LIN {X 0,Y 375.167,Z 691.382,A -85,B 0,C 180,E1 -12319.202,E2 -12319.202} C_VEL
LIN {X 0,Y 374.786,Z 697.005,A -85,B 0,C 180,E1 -12321.371,E2 -12321.371} C_VEL
LIN {X 0,Y 374.563,Z 701.231,A -85,B 0,C 180,E1 -12323.534,E2 -12323.534} C_VEL
LIN {X 0,Y 374.483,Z 704.148,A -85,B 0,C 180,E1 -12325.693,E2 -12325.693} C_VEL
LIN {X 0,Y 374.459,Z 705.82,A -85,B 0,C 180,E1 -12327.847,E2 -12327.847} C_VEL
LIN {X 0,Y 374.551,Z 706.272,A -85,B 0,C 180,E1 -12329.998,E2 -12329.998} C_VEL
LIN {X 0,Y 374.492,Z 705.492,A -85,B 0,C 180,E1 -12332.149,E2 -12332.149} C_VEL
LIN {X 0,Y 374.518,Z 703.472,A -85,B 0,C 180,E1 -12334.303,E2 -12334.303} C_VEL
LIN {X 0,Y 374.568,Z 700.142,A -85,B 0,C 180,E1 -12336.462,E2 -12336.462} C_VEL
LIN {X 0,Y 374.757,Z 695.441,A -85,B 0,C 180,E1 -12338.627,E2 -12338.627} C_VEL
LIN {X 0,Y 375.119,Z 689.261,A -85,B 0,C 180,E1 -12340.797,E2 -12340.797} C_VEL
LIN {X 0,Y 375.816,Z 681.448,A -85,B 0,C 180,E1 -12342.966,E2 -12342.966} C_VEL
LIN {X 0,Y 376.604,Z 673.027,A -85,B 0,C 180,E1 -12344.866,E2 -12344.866} C_VEL
LIN {X 0,Y 377.653,Z 662.889,A -85,B 0,C 180,E1 -12346.763,E2 -12346.763} C_VEL
LIN {X 0,Y 378.997,Z 651.186,A -85,B 0,C 180,E1 -12348.568,E2 -12348.568} C_VEL
LIN {X 0,Y 380.268,Z 638.932,A -85,B 0,C 180,E1 -12350.132,E2 -12350.132} C_VEL
LIN {X 0,Y 381.757,Z 626.326,A -85,B 0,C 180,E1 -12351.46,E2 -12351.46} C_VEL
LIN {X 0,Y 383.095,Z 612.535,A -85,B 0,C 180,E1 -12352.657,E2 -12352.657} C_VEL
LIN {X 0,Y 384.47,Z 598.386,A -85,B 0,C 180,E1 -12353.639,E2 -12353.639} C_VEL
LIN {X 0,Y 385.599,Z 583.226,A -85,B 0,C 180,E1 -12354.461,E2 -12354.461} C_VEL
LIN {X 0,Y 386.578,Z 567.645,A -85,B 0,C 180,E1 -12355.074,E2 -12355.074} C_VEL
LIN {X 0,Y 387.201,Z 551.46,A -85,B 0,C 180,E1 -12355.498,E2 -12355.498} C_VEL
LIN {X 0,Y 390.699,Z 433.656,A -85,B 0,C 180,E1 -12358.035,E2 -12358.035} C_VEL
LIN {X 0,Y 384.578,Z 400.558,A -85,B 0,C 180,E1 -12359.257,E2 -12359.257} C_VEL
LIN {X 0,Y 382.474,Z 394.871,A -85,B 0,C 180,E1 -12359.562,E2 -12359.562} C_VEL
LIN {X 0,Y 378.805,Z 379.595,A -85,B 0,C 180,E1 -12362.771,E2 -12362.771} C_VEL
LIN {X 0,Y 376.004,Z 368.274,A -85,B 0,C 180,E1 -12365.309,E2 -12365.309} C_VEL
LIN {X 0,Y 375.925,Z 368.286,A -85,B 0,C 180,E1 -12368.261,E2 -12368.261} C_VEL
LIN {X 0,Y 375.907,Z 368.283,A -85,B 0,C 180,E1 -12371.596,E2 -12371.596} C_VEL
LIN {X 0,Y 375.913,Z 368.282,A -85,B 0,C 180,E1 -12374.73,E2 -12374.73} C_VEL
LIN {X 0,Y 375.914,Z 368.283,A -85,B 0,C 180,E1 -12377.698,E2 -12377.698} C_VEL
LIN {X 0,Y 375.921,Z 368.283,A -85,B 0,C 180,E1 -12380.533,E2 -12380.533} C_VEL
LIN {X 0,Y 375.946,Z 368.277,A -85,B 0,C 180,E1 -12383.496,E2 -12383.496} C_VEL
LIN {X 0,Y 375.946,Z 368.281,A -85,B 0,C 180,E1 -12385.887,E2 -12385.887} C_VEL
LIN {X 0,Y 375.948,Z 368.279,A -85,B 0,C 180,E1 -12389.686,E2 -12389.686} C_VEL
LIN {X 0,Y 375.904,Z 368.289,A -85,B 0,C 180,E1 -12392.134,E2 -12392.134} C_VEL
LIN {X 0,Y 375.921,Z 368.282,A -85,B 0,C 180,E1 -12394.533,E2 -12394.533} C_VEL
LIN {X 0,Y 375.959,Z 368.275,A -85,B 0,C 180,E1 -12396.886,E2 -12396.886} C_VEL
LIN {X 0,Y 375.98,Z 368.276,A -85,B 0,C 180,E1 -12400.339,E2 -12400.339} C_VEL
LIN {X 0,Y 375.96,Z 368.278,A -85,B 0,C 180,E1 -12403.716,E2 -12403.716} C_VEL
LIN {X 0,Y 376.089,Z 368.259,A -85,B 0,C 180,E1 -12407.042,E2 -12407.042} C_VEL
LIN {X 0,Y 376.097,Z 368.262,A -85,B 0,C 180,E1 -12410.318,E2 -12410.318} C_VEL
LIN {X 0,Y 376.183,Z 368.249,A -85,B 0,C 180,E1 -12413.564,E2 -12413.564} C_VEL
LIN {X 0,Y 376.322,Z 368.235,A -85,B 0,C 180,E1 -12417.86,E2 -12417.86} C_VEL
LIN {X 0,Y 376.215,Z 368.243,A -85,B 0,C 180,E1 -12421.071,E2 -12421.071} C_VEL
LIN {X 0,Y 376.322,Z 368.235,A -85,B 0,C 180,E1 -12422.141,E2 -12422.141} C_VEL
LIN {X 0,Y 376.18,Z 368.249,A -85,B 0,C 180,E1 -12426.46,E2 -12426.46} C_VEL
LIN {X 0,Y 376.093,Z 368.262,A -85,B 0,C 180,E1 -12429.682,E2 -12429.682} C_VEL
LIN {X 0,Y 376.076,Z 368.264,A -85,B 0,C 180,E1 -12433.658,E2 -12433.658} C_VEL
LIN {X 0,Y 375.998,Z 368.273,A -85,B 0,C 180,E1 -12437.592,E2 -12437.592} C_VEL
LIN {X 0,Y 375.966,Z 368.274,A -85,B 0,C 180,E1 -12440.833,E2 -12440.833} C_VEL
LIN {X 0,Y 375.923,Z 368.282,A -85,B 0,C 180,E1 -12444.287,E2 -12444.287} C_VEL
LIN {X 0,Y 375.899,Z 368.283,A -85,B 0,C 180,E1 -12446.662,E2 -12446.662} C_VEL
LIN {X 0,Y 375.902,Z 368.282,A -85,B 0,C 180,E1 -12449.085,E2 -12449.085} C_VEL
LIN {X 0,Y 375.946,Z 368.28,A -85,B 0,C 180,E1 -12451.563,E2 -12451.563} C_VEL
LIN {X 0,Y 375.941,Z 368.279,A -85,B 0,C 180,E1 -12455.418,E2 -12455.418} C_VEL
LIN {X 0,Y 375.924,Z 368.282,A -85,B 0,C 180,E1 -12458.264,E2 -12458.264} C_VEL
LIN {X 0,Y 375.907,Z 368.285,A -85,B 0,C 180,E1 -12461.599,E2 -12461.599} C_VEL
LIN {X 0,Y 375.914,Z 368.281,A -85,B 0,C 180,E1 -12464.732,E2 -12464.732} C_VEL
LIN {X 0,Y 375.908,Z 368.287,A -85,B 0,C 180,E1 -12467.699,E2 -12467.699} C_VEL
LIN {X 0,Y 375.927,Z 368.28,A -85,B 0,C 180,E1 -12470.536,E2 -12470.536} C_VEL
LIN {X 0,Y 375.952,Z 368.279,A -85,B 0,C 180,E1 -12473.499,E2 -12473.499} C_VEL
LIN {X 0,Y 375.953,Z 368.281,A -85,B 0,C 180,E1 -12475.89,E2 -12475.89} C_VEL
LIN {X 0,Y 375.957,Z 368.281,A -85,B 0,C 180,E1 -12479.689,E2 -12479.689} C_VEL
LIN {X 0,Y 375.914,Z 368.283,A -85,B 0,C 180,E1 -12482.137,E2 -12482.137} C_VEL
LIN {X 0,Y 375.956,Z 368.282,A -85,B 0,C 180,E1 -12485.718,E2 -12485.718} C_VEL
LIN {X 0,Y 375.997,Z 368.272,A -85,B 0,C 180,E1 -12489.2,E2 -12489.2} C_VEL
LIN {X 0,Y 376.032,Z 368.266,A -85,B 0,C 180,E1 -12492.602,E2 -12492.602} C_VEL
LIN {X 0,Y 376.09,Z 368.26,A -85,B 0,C 180,E1 -12496.344,E2 -12496.344} C_VEL
LIN {X 0,Y 376.114,Z 368.257,A -85,B 0,C 180,E1 -12500.32,E2 -12500.32} C_VEL
LIN {X 0,Y 376.195,Z 368.251,A -85,B 0,C 180,E1 -12503.566,E2 -12503.566} C_VEL
LIN {X 0,Y 376.34,Z 368.232,A -85,B 0,C 180,E1 -12507.861,E2 -12507.861} C_VEL
LIN {X 0,Y 376.235,Z 368.242,A -85,B 0,C 180,E1 -12511.072,E2 -12511.072} C_VEL
LIN {X 0,Y 376.342,Z 368.229,A -85,B 0,C 180,E1 -12512.142,E2 -12512.142} C_VEL
LIN {X 0,Y 376.203,Z 368.245,A -85,B 0,C 180,E1 -12516.437,E2 -12516.437} C_VEL
LIN {X 0,Y 376.118,Z 368.261,A -85,B 0,C 180,E1 -12519.683,E2 -12519.683} C_VEL
LIN {X 0,Y 376.095,Z 368.264,A -85,B 0,C 180,E1 -12523.659,E2 -12523.659} C_VEL
LIN {X 0,Y 376.014,Z 368.275,A -85,B 0,C 180,E1 -12527.591,E2 -12527.591} C_VEL
LIN {X 0,Y 375.985,Z 368.272,A -85,B 0,C 180,E1 -12530.833,E2 -12530.833} C_VEL
LIN {X 0,Y 375.941,Z 368.278,A -85,B 0,C 180,E1 -12534.286,E2 -12534.286} C_VEL
LIN {X 0,Y 375.925,Z 368.279,A -85,B 0,C 180,E1 -12536.661,E2 -12536.661} C_VEL
LIN {X 0,Y 375.922,Z 368.282,A -85,B 0,C 180,E1 -12539.085,E2 -12539.085} C_VEL
LIN {X 0,Y 375.964,Z 368.281,A -85,B 0,C 180,E1 -12541.563,E2 -12541.563} C_VEL
LIN {X 0,Y 375.964,Z 368.28,A -85,B 0,C 180,E1 -12545.416,E2 -12545.416} C_VEL
LIN {X 0,Y 375.939,Z 368.28,A -85,B 0,C 180,E1 -12548.379,E2 -12548.379} C_VEL
LIN {X 0,Y 375.802,Z 368.937,A -85,B 0,C 180,E1 -12548.942,E2 -12548.942} C_VEL
LIN {X 0,Y 375.457,Z 371.132,A -85,B 0,C 180,E1 -12549.583,E2 -12549.583} C_VEL
LIN {X 0,Y 375.103,Z 374.321,A -85,B 0,C 180,E1 -12550.139,E2 -12550.139} C_VEL
LIN {X 0,Y 374.91,Z 379.094,A -85,B 0,C 180,E1 -12550.703,E2 -12550.703} C_VEL
LIN {X 0,Y 375.28,Z 384.418,A -85,B 0,C 180,E1 -12551.165,E2 -12551.165} C_VEL
LIN {X 0,Y 376.697,Z 389.883,A -85,B 0,C 180,E1 -12551.517,E2 -12551.517} C_VEL
LIN {X 0,Y 384.508,Z 409.226,A -85,B 0,C 180,E1 -12552.555,E2 -12552.555} C_VEL
LIN {X 0,Y 380.344,Z 540.89,A -85,B 0,C 180,E1 -12555.483,E2 -12555.483} C_VEL
LIN {X 0,Y 379.526,Z 556.254,A -85,B 0,C 180,E1 -12556.027,E2 -12556.027} C_VEL
LIN {X 0,Y 378.509,Z 571.5,A -85,B 0,C 180,E1 -12556.789,E2 -12556.789} C_VEL
LIN {X 0,Y 377.323,Z 585.701,A -85,B 0,C 180,E1 -12557.711,E2 -12557.711} C_VEL
LIN {X 0,Y 376.012,Z 599.504,A -85,B 0,C 180,E1 -12558.834,E2 -12558.834} C_VEL
LIN {X 0,Y 374.683,Z 612.193,A -85,B 0,C 180,E1 -12560.093,E2 -12560.093} C_VEL
LIN {X 0,Y 373.27,Z 624.646,A -85,B 0,C 180,E1 -12561.586,E2 -12561.586} C_VEL
LIN {X 0,Y 371.958,Z 635.478,A -85,B 0,C 180,E1 -12563.136,E2 -12563.136} C_VEL
LIN {X 0,Y 370.845,Z 645.284,A -85,B 0,C 180,E1 -12564.811,E2 -12564.811} C_VEL
LIN {X 0,Y 369.765,Z 654.806,A -85,B 0,C 180,E1 -12566.753,E2 -12566.753} C_VEL
LIN {X 0,Y 368.928,Z 662.904,A -85,B 0,C 180,E1 -12568.759,E2 -12568.759} C_VEL
LIN {X 0,Y 368.304,Z 669.864,A -85,B 0,C 180,E1 -12570.883,E2 -12570.883} C_VEL
LIN {X 0,Y 367.929,Z 674.668,A -85,B 0,C 180,E1 -12572.713,E2 -12572.713} C_VEL
LIN {X 0,Y 367.613,Z 678.523,A -85,B 0,C 180,E1 -12574.533,E2 -12574.533} C_VEL
LIN {X 0,Y 367.356,Z 681.852,A -85,B 0,C 180,E1 -12576.682,E2 -12576.682} C_VEL
LIN {X 0,Y 367.204,Z 683.837,A -85,B 0,C 180,E1 -12578.675,E2 -12578.675} C_VEL
LIN {X 0,Y 367.261,Z 684.548,A -85,B 0,C 180,E1 -12579.851,E2 -12579.851} C_VEL
LIN {X 0,Y 367.214,Z 684.935,A -85,B 0,C 180,E1 -12582.168,E2 -12582.168} C_VEL
LIN {X 0,Y 367.311,Z 683.991,A -85,B 0,C 180,E1 -12584.462,E2 -12584.462} C_VEL
LIN {X 0,Y 367.532,Z 681.758,A -85,B 0,C 180,E1 -12586.734,E2 -12586.734} C_VEL
LIN {X 0,Y 367.936,Z 678.221,A -85,B 0,C 180,E1 -12588.988,E2 -12588.988} C_VEL
LIN {X 0,Y 368.482,Z 673.342,A -85,B 0,C 180,E1 -12591.223,E2 -12591.223} C_VEL
LIN {X 0,Y 369.331,Z 667.002,A -85,B 0,C 180,E1 -12593.444,E2 -12593.444} C_VEL
LIN {X 0,Y 370.475,Z 659.049,A -85,B 0,C 180,E1 -12595.648,E2 -12595.648} C_VEL
LIN {X 0,Y 371.712,Z 650.629,A -85,B 0,C 180,E1 -12597.562,E2 -12597.562} C_VEL
LIN {X 0,Y 373.077,Z 641.973,A -85,B 0,C 180,E1 -12599.21,E2 -12599.21} C_VEL
LIN {X 0,Y 374.527,Z 632.037,A -85,B 0,C 180,E1 -12600.806,E2 -12600.806} C_VEL
LIN {X 0,Y 376.314,Z 620.105,A -85,B 0,C 180,E1 -12602.408,E2 -12602.408} C_VEL
LIN {X 0,Y 378.203,Z 607.026,A -85,B 0,C 180,E1 -12603.862,E2 -12603.862} C_VEL
LIN {X 0,Y 379.83,Z 594.125,A -85,B 0,C 180,E1 -12605.042,E2 -12605.042} C_VEL
LIN {X 0,Y 381.38,Z 580.116,A -85,B 0,C 180,E1 -12606.082,E2 -12606.082} C_VEL
LIN {X 0,Y 382.788,Z 565.599,A -85,B 0,C 180,E1 -12606.926,E2 -12606.926} C_VEL
LIN {X 0,Y 383.995,Z 549.612,A -85,B 0,C 180,E1 -12607.625,E2 -12607.625} C_VEL
LIN {X 0,Y 384.909,Z 532.197,A -85,B 0,C 180,E1 -12608.135,E2 -12608.135} C_VEL
LIN {X 0,Y 389.101,Z 444.121,A -85,B 0,C 180,E1 -12610.286,E2 -12610.286} C_VEL
LIN {X 0,Y 390.641,Z 413.247,A -85,B 0,C 180,E1 -12611.082,E2 -12611.082} C_VEL
LIN {X 0,Y 385.442,Z 401.984,A -85,B 0,C 180,E1 -12612.085,E2 -12612.085} C_VEL
LIN {X 0,Y 377.727,Z 387.787,A -85,B 0,C 180,E1 -12613.643,E2 -12613.643} C_VEL
LIN {X 0,Y 373.949,Z 381.999,A -85,B 0,C 180,E1 -12614.434,E2 -12614.434} C_VEL
LIN {X 0,Y 372.106,Z 378.757,A -85,B 0,C 180,E1 -12614.895,E2 -12614.895} C_VEL
LIN {X 0,Y 369.71,Z 371.508,A -85,B 0,C 180,E1 -12617.707,E2 -12617.707} C_VEL
LIN {X 0,Y 368.973,Z 369.151,A -85,B 0,C 180,E1 -12618.735,E2 -12618.735} C_VEL
LIN {X 0,Y 368.904,Z 369.159,A -85,B 0,C 180,E1 -12622.397,E2 -12622.397} C_VEL
LIN {X 0,Y 368.924,Z 369.157,A -85,B 0,C 180,E1 -12625.986,E2 -12625.986} C_VEL
LIN {X 0,Y 368.897,Z 369.158,A -85,B 0,C 180,E1 -12629.692,E2 -12629.692} C_VEL
LIN {X 0,Y 368.9,Z 369.157,A -85,B 0,C 180,E1 -12633.042,E2 -12633.042} C_VEL
LIN {X 0,Y 368.914,Z 369.157,A -85,B 0,C 180,E1 -12636.197,E2 -12636.197} C_VEL
LIN {X 0,Y 368.876,Z 369.16,A -85,B 0,C 180,E1 -12638.956,E2 -12638.956} C_VEL
LIN {X 0,Y 368.861,Z 369.161,A -85,B 0,C 180,E1 -12642.004,E2 -12642.004} C_VEL
LIN {X 0,Y 368.875,Z 369.158,A -85,B 0,C 180,E1 -12645.173,E2 -12645.173} C_VEL
LIN {X 0,Y 368.877,Z 369.159,A -85,B 0,C 180,E1 -12648.904,E2 -12648.904} C_VEL
LIN {X 0,Y 368.913,Z 369.309,A -85,B 0,C 180,E1 -12649.27,E2 -12649.27} C_VEL
LIN {X 0,Y 371.502,Z 376.86,A -85,B 0,C 180,E1 -12652.168,E2 -12652.168} C_VEL
LIN {X 0,Y 373.882,Z 384.509,A -85,B 0,C 180,E1 -12654.688,E2 -12654.688} C_VEL
LIN {X 0,Y 375.91,Z 391.786,A -85,B 0,C 180,E1 -12656.771,E2 -12656.771} C_VEL
LIN {X 0,Y 381.445,Z 402.585,A -85,B 0,C 180,E1 -12657.944,E2 -12657.944} C_VEL
LIN {X 0,Y 386.148,Z 412.739,A -85,B 0,C 180,E1 -12658.901,E2 -12658.901} C_VEL
LIN {X 0,Y 388.976,Z 429.056,A -85,B 0,C 180,E1 -12659.765,E2 -12659.765} C_VEL
LIN {X 0,Y 389.905,Z 436.075,A -85,B 0,C 180,E1 -12660.095,E2 -12660.095} C_VEL
LIN {X 0,Y 385.058,Z 537.741,A -85,B 0,C 180,E1 -12662.593,E2 -12662.593} C_VEL
LIN {X 0,Y 383.828,Z 562.645,A -85,B 0,C 180,E1 -12663.234,E2 -12663.234} C_VEL
LIN {X 0,Y 382.507,Z 579.171,A -85,B 0,C 180,E1 -12663.87,E2 -12663.87} C_VEL
LIN {X 0,Y 381.081,Z 593.255,A -85,B 0,C 180,E1 -12664.609,E2 -12664.609} C_VEL
LIN {X 0,Y 379.44,Z 607.638,A -85,B 0,C 180,E1 -12665.58,E2 -12665.58} C_VEL
LIN {X 0,Y 377.957,Z 619.65,A -85,B 0,C 180,E1 -12666.579,E2 -12666.579} C_VEL
LIN {X 0,Y 376.092,Z 632.901,A -85,B 0,C 180,E1 -12667.908,E2 -12667.908} C_VEL
LIN {X 0,Y 374.316,Z 645.16,A -85,B 0,C 180,E1 -12669.386,E2 -12669.386} C_VEL
LIN {X 0,Y 372.633,Z 656.795,A -85,B 0,C 180,E1 -12671.076,E2 -12671.076} C_VEL
LIN {X 0,Y 371.095,Z 667.393,A -85,B 0,C 180,E1 -12672.928,E2 -12672.928} C_VEL
LIN {X 0,Y 369.831,Z 676.544,A -85,B 0,C 180,E1 -12674.852,E2 -12674.852} C_VEL
LIN {X 0,Y 368.899,Z 684.222,A -85,B 0,C 180,E1 -12676.783,E2 -12676.783} C_VEL
LIN {X 0,Y 368.147,Z 691.339,A -85,B 0,C 180,E1 -12678.993,E2 -12678.993} C_VEL
LIN {X 0,Y 367.724,Z 696.933,A -85,B 0,C 180,E1 -12681.204,E2 -12681.204} C_VEL
LIN {X 0,Y 367.481,Z 701.121,A -85,B 0,C 180,E1 -12683.409,E2 -12683.409} C_VEL
LIN {X 0,Y 367.391,Z 704.002,A -85,B 0,C 180,E1 -12685.61,E2 -12685.61} C_VEL
LIN {X 0,Y 367.358,Z 705.636,A -85,B 0,C 180,E1 -12687.806,E2 -12687.806} C_VEL
LIN {X 0,Y 367.454,Z 706.05,A -85,B 0,C 180,E1 -12689.998,E2 -12689.998} C_VEL
LIN {X 0,Y 367.392,Z 705.228,A -85,B 0,C 180,E1 -12692.191,E2 -12692.191} C_VEL
LIN {X 0,Y 367.423,Z 703.164,A -85,B 0,C 180,E1 -12694.386,E2 -12694.386} C_VEL
LIN {X 0,Y 367.488,Z 699.799,A -85,B 0,C 180,E1 -12696.587,E2 -12696.587} C_VEL
LIN {X 0,Y 367.7,Z 695.045,A -85,B 0,C 180,E1 -12698.794,E2 -12698.794} C_VEL
LIN {X 0,Y 368.094,Z 688.799,A -85,B 0,C 180,E1 -12701.005,E2 -12701.005} C_VEL
LIN {X 0,Y 368.774,Z 680.896,A -85,B 0,C 180,E1 -12703.218,E2 -12703.218} C_VEL
LIN {X 0,Y 369.649,Z 672.404,A -85,B 0,C 180,E1 -12705.153,E2 -12705.153} C_VEL
LIN {X 0,Y 370.773,Z 662.154,A -85,B 0,C 180,E1 -12707.084,E2 -12707.084} C_VEL
LIN {X 0,Y 372.007,Z 651.643,A -85,B 0,C 180,E1 -12708.732,E2 -12708.732} C_VEL
LIN {X 0,Y 373.371,Z 639.077,A -85,B 0,C 180,E1 -12710.377,E2 -12710.377} C_VEL
LIN {X 0,Y 374.899,Z 626.524,A -85,B 0,C 180,E1 -12711.728,E2 -12711.728} C_VEL
LIN {X 0,Y 376.269,Z 612.818,A -85,B 0,C 180,E1 -12712.947,E2 -12712.947} C_VEL
LIN {X 0,Y 377.686,Z 598.79,A -85,B 0,C 180,E1 -12713.945,E2 -12713.945} C_VEL
LIN {X 0,Y 378.867,Z 583.97,A -85,B 0,C 180,E1 -12714.773,E2 -12714.773} C_VEL
LIN {X 0,Y 379.854,Z 568.68,A -85,B 0,C 180,E1 -12715.403,E2 -12715.403} C_VEL
LIN {X 0,Y 380.51,Z 553.188,A -85,B 0,C 180,E1 -12715.833,E2 -12715.833} C_VEL
LIN {X 0,Y 384.165,Z 434.608,A -85,B 0,C 180,E1 -12718.448,E2 -12718.448} C_VEL
LIN {X 0,Y 378.379,Z 403.023,A -85,B 0,C 180,E1 -12719.636,E2 -12719.636} C_VEL
LIN {X 0,Y 375.175,Z 394.648,A -85,B 0,C 180,E1 -12720.105,E2 -12720.105} C_VEL
LIN {X 0,Y 371.675,Z 379.983,A -85,B 0,C 180,E1 -12723.252,E2 -12723.252} C_VEL
LIN {X 0,Y 368.928,Z 369.157,A -85,B 0,C 180,E1 -12725.735,E2 -12725.735} C_VEL
LIN {X 0,Y 368.863,Z 369.163,A -85,B 0,C 180,E1 -12728.956,E2 -12728.956} C_VEL
LIN {X 0,Y 368.86,Z 369.164,A -85,B 0,C 180,E1 -12732.006,E2 -12732.006} C_VEL
LIN {X 0,Y 368.866,Z 369.159,A -85,B 0,C 180,E1 -12735.174,E2 -12735.174} C_VEL
LIN {X 0,Y 368.857,Z 369.167,A -85,B 0,C 180,E1 -12738.174,E2 -12738.174} C_VEL
LIN {X 0,Y 368.863,Z 369.159,A -85,B 0,C 180,E1 -12741.365,E2 -12741.365} C_VEL
LIN {X 0,Y 368.92,Z 369.152,A -85,B 0,C 180,E1 -12745.145,E2 -12745.145} C_VEL
LIN {X 0,Y 368.899,Z 369.155,A -85,B 0,C 180,E1 -12749.044,E2 -12749.044} C_VEL
LIN {X 0,Y 368.893,Z 369.157,A -85,B 0,C 180,E1 -12751.557,E2 -12751.557} C_VEL
LIN {X 0,Y 368.872,Z 369.158,A -85,B 0,C 180,E1 -12755.219,E2 -12755.219} C_VEL
LIN {X 0,Y 368.884,Z 369.158,A -85,B 0,C 180,E1 -12757.602,E2 -12757.602} C_VEL
LIN {X 0,Y 368.921,Z 369.152,A -85,B 0,C 180,E1 -12761.104,E2 -12761.104} C_VEL
LIN {X 0,Y 368.925,Z 369.153,A -85,B 0,C 180,E1 -12764.532,E2 -12764.532} C_VEL
LIN {X 0,Y 369.043,Z 369.137,A -85,B 0,C 180,E1 -12766.79,E2 -12766.79} C_VEL
LIN {X 0,Y 369.047,Z 369.142,A -85,B 0,C 180,E1 -12770.131,E2 -12770.131} C_VEL
LIN {X 0,Y 369.144,Z 369.125,A -85,B 0,C 180,E1 -12773.441,E2 -12773.441} C_VEL
LIN {X 0,Y 369.286,Z 369.111,A -85,B 0,C 180,E1 -12777.819,E2 -12777.819} C_VEL
LIN {X 0,Y 369.187,Z 369.119,A -85,B 0,C 180,E1 -12781.091,E2 -12781.091} C_VEL
LIN {X 0,Y 369.285,Z 369.111,A -85,B 0,C 180,E1 -12782.182,E2 -12782.182} C_VEL
LIN {X 0,Y 369.143,Z 369.125,A -85,B 0,C 180,E1 -12786.56,E2 -12786.56} C_VEL
LIN {X 0,Y 369.044,Z 369.142,A -85,B 0,C 180,E1 -12789.869,E2 -12789.869} C_VEL
LIN {X 0,Y 369.023,Z 369.144,A -85,B 0,C 180,E1 -12793.773,E2 -12793.773} C_VEL
LIN {X 0,Y 368.964,Z 369.151,A -85,B 0,C 180,E1 -12797.758,E2 -12797.758} C_VEL
LIN {X 0,Y 368.896,Z 369.155,A -85,B 0,C 180,E1 -12801.222,E2 -12801.222} C_VEL
LIN {X 0,Y 368.898,Z 369.161,A -85,B 0,C 180,E1 -12803.876,E2 -12803.876} C_VEL
LIN {X 0,Y 368.845,Z 369.162,A -85,B 0,C 180,E1 -12807.213,E2 -12807.213} C_VEL
LIN {X 0,Y 368.881,Z 369.161,A -85,B 0,C 180,E1 -12809.694,E2 -12809.694} C_VEL
LIN {X 0,Y 368.886,Z 369.156,A -85,B 0,C 180,E1 -12813.045,E2 -12813.045} C_VEL
LIN {X 0,Y 368.902,Z 369.157,A -85,B 0,C 180,E1 -12816.199,E2 -12816.199} C_VEL
LIN {X 0,Y 368.863,Z 369.159,A -85,B 0,C 180,E1 -12818.959,E2 -12818.959} C_VEL
LIN {X 0,Y 368.861,Z 369.164,A -85,B 0,C 180,E1 -12822.009,E2 -12822.009} C_VEL
LIN {X 0,Y 368.866,Z 369.159,A -85,B 0,C 180,E1 -12825.177,E2 -12825.177} C_VEL
LIN {X 0,Y 368.857,Z 369.163,A -85,B 0,C 180,E1 -12828.177,E2 -12828.177} C_VEL
LIN {X 0,Y 368.869,Z 369.16,A -85,B 0,C 180,E1 -12831.368,E2 -12831.368} C_VEL
LIN {X 0,Y 368.925,Z 369.152,A -85,B 0,C 180,E1 -12835.148,E2 -12835.148} C_VEL
LIN {X 0,Y 368.908,Z 369.154,A -85,B 0,C 180,E1 -12839.047,E2 -12839.047} C_VEL
LIN {X 0,Y 368.903,Z 369.158,A -85,B 0,C 180,E1 -12841.56,E2 -12841.56} C_VEL
LIN {X 0,Y 368.895,Z 369.157,A -85,B 0,C 180,E1 -12845.222,E2 -12845.222} C_VEL
LIN {X 0,Y 368.918,Z 369.157,A -85,B 0,C 180,E1 -12847.606,E2 -12847.606} C_VEL
LIN {X 0,Y 368.953,Z 369.149,A -85,B 0,C 180,E1 -12851.108,E2 -12851.108} C_VEL
LIN {X 0,Y 368.997,Z 369.143,A -85,B 0,C 180,E1 -12854.537,E2 -12854.537} C_VEL
LIN {X 0,Y 369.005,Z 369.146,A -85,B 0,C 180,E1 -12857.909,E2 -12857.909} C_VEL
LIN {X 0,Y 369.092,Z 369.133,A -85,B 0,C 180,E1 -12861.24,E2 -12861.24} C_VEL
LIN {X 0,Y 369.118,Z 369.127,A -85,B 0,C 180,E1 -12864.539,E2 -12864.539} C_VEL
LIN {X 0,Y 369.304,Z 369.109,A -85,B 0,C 180,E1 -12867.82,E2 -12867.82} C_VEL
LIN {X 0,Y 369.206,Z 369.118,A -85,B 0,C 180,E1 -12871.092,E2 -12871.092} C_VEL
LIN {X 0,Y 369.306,Z 369.105,A -85,B 0,C 180,E1 -12872.183,E2 -12872.183} C_VEL
LIN {X 0,Y 369.163,Z 369.122,A -85,B 0,C 180,E1 -12876.561,E2 -12876.561} C_VEL
LIN {X 0,Y 369.068,Z 369.137,A -85,B 0,C 180,E1 -12879.87,E2 -12879.87} C_VEL
LIN {X 0,Y 369.043,Z 369.141,A -85,B 0,C 180,E1 -12883.774,E2 -12883.774} C_VEL
LIN {X 0,Y 368.959,Z 369.152,A -85,B 0,C 180,E1 -12887.746,E2 -12887.746} C_VEL
LIN {X 0,Y 368.935,Z 369.153,A -85,B 0,C 180,E1 -12891.221,E2 -12891.221} C_VEL
LIN {X 0,Y 368.916,Z 369.156,A -85,B 0,C 180,E1 -12893.876,E2 -12893.876} C_VEL
LIN {X 0,Y 368.87,Z 369.161,A -85,B 0,C 180,E1 -12897.212,E2 -12897.212} C_VEL
LIN {X 0,Y 368.936,Z 369.151,A -85,B 0,C 180,E1 -12900.954,E2 -12900.954} C_VEL
LIN {X 0,Y 368.935,Z 369.152,A -85,B 0,C 180,E1 -12905.002,E2 -12905.002} C_VEL
LIN {X 0,Y 368.896,Z 369.16,A -85,B 0,C 180,E1 -12908.637,E2 -12908.637} C_VEL
LIN {X 0,Y 368.919,Z 369.19,A -85,B 0,C 180,E1 -12909.304,E2 -12909.304} C_VEL
LIN {X 0,Y 370.294,Z 374.913,A -85,B 0,C 180,E1 -12910.658,E2 -12910.658} C_VEL
LIN {X 0,Y 376.697,Z 389.883,A -85,B 0,C 180,E1 -12911.517,E2 -12911.517} C_VEL
LIN {X 0,Y 378.187,Z 395.394,A -85,B 0,C 180,E1 -12911.765,E2 -12911.765} C_VEL
LIN {X 0,Y 378.729,Z 401.209,A -85,B 0,C 180,E1 -12911.951,E2 -12911.951} C_VEL
LIN {X 0,Y 378.185,Z 413.221,A -85,B 0,C 180,E1 -12912.215,E2 -12912.215} C_VEL
LIN {X 0,Y 377.658,Z 421.248,A -85,B 0,C 180,E1 -12912.381,E2 -12912.381} C_VEL
LIN {X 0,Y 373.71,Z 541.148,A -85,B 0,C 180,E1 -12915.104,E2 -12915.104} C_VEL
LIN {X 0,Y 372.859,Z 556.542,A -85,B 0,C 180,E1 -12915.662,E2 -12915.662} C_VEL
LIN {X 0,Y 371.866,Z 570.887,A -85,B 0,C 180,E1 -12916.383,E2 -12916.383} C_VEL
LIN {X 0,Y 370.587,Z 585.96,A -85,B 0,C 180,E1 -12917.377,E2 -12917.377} C_VEL
LIN {X 0,Y 369.148,Z 600.394,A -85,B 0,C 180,E1 -12918.579,E2 -12918.579} C_VEL
LIN {X 0,Y 367.71,Z 613.727,A -85,B 0,C 180,E1 -12919.948,E2 -12919.948} C_VEL
LIN {X 0,Y 366.292,Z 625.64,A -85,B 0,C 180,E1 -12921.423,E2 -12921.423} C_VEL
LIN {X 0,Y 364.952,Z 636.357,A -85,B 0,C 180,E1 -12923.001,E2 -12923.001} C_VEL
LIN {X 0,Y 363.697,Z 647.113,A -85,B 0,C 180,E1 -12924.908,E2 -12924.908} C_VEL
LIN {X 0,Y 362.68,Z 655.834,A -85,B 0,C 180,E1 -12926.76,E2 -12926.76} C_VEL
LIN {X 0,Y 361.854,Z 663.487,A -85,B 0,C 180,E1 -12928.715,E2 -12928.715} C_VEL
